Yaskawa INFORM job: DEMO_ROOF_SIDE_0625_3PAINT_2.JBI

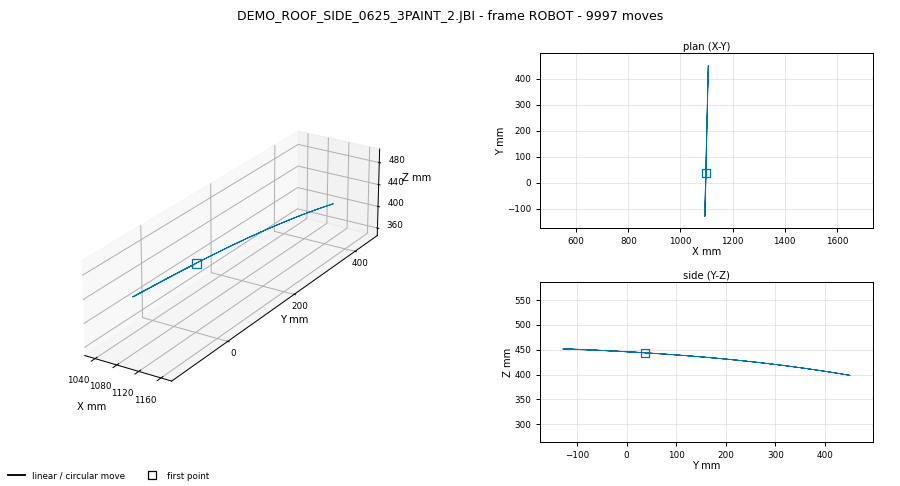
[picture p0: tool path of DEMO_ROOF_SIDE_0625_3PAINT_2.JBI in frame ROBOT, 9997 of 9997 moves have a stored position in this frame; points joined in program order, loops and branches not executed]
/JOB
//NAME DEMO_ROOF_SIDE_0625_3PAINT2
//POS
///NPOS 9997,0,0,0,0,0
///TOOL 0
///USER 0
///POSTYPE ROBOT
///RECTAN
///RCONF 1,0,0,0,0,0,0,0,0,0,0,0,0,0,0,0,0,0,0,0,0,0,0,0
C00000=1098.370,36.999,444.195,176.206,15.311,152.033
C00001=1098.365,36.749,444.210,176.204,15.310,152.034
C00002=1098.358,36.500,444.225,176.201,15.310,152.034
C00003=1098.353,36.250,444.240,176.199,15.308,152.034
C00004=1098.347,36.001,444.255,176.197,15.308,152.035
C00005=1098.341,35.751,444.271,176.195,15.307,152.035
C00006=1098.336,35.502,444.287,176.192,15.306,152.035
C00007=1098.329,35.252,444.302,176.190,15.306,152.036
C00008=1098.324,35.003,444.317,176.188,15.305,152.036
C00009=1098.318,34.753,444.332,176.185,15.304,152.036
C00010=1098.312,34.503,444.347,176.183,15.303,152.037
C00011=1098.307,34.255,444.362,176.181,15.303,152.037
C00012=1098.301,34.005,444.377,176.178,15.302,152.037
C00013=1098.296,33.755,444.393,176.176,15.301,152.038
C00014=1098.289,33.506,444.407,176.174,15.301,152.038
C00015=1098.284,33.256,444.423,176.172,15.300,152.038
C00016=1098.278,33.007,444.438,176.170,15.299,152.038
C00017=1098.273,32.758,444.453,176.167,15.298,152.039
C00018=1098.266,32.508,444.468,176.166,15.298,152.039
C00019=1098.261,32.258,444.484,176.163,15.296,152.039
C00020=1098.254,31.985,444.500,176.161,15.296,152.040
C00021=1098.248,31.711,444.517,176.158,15.295,152.040
C00022=1098.242,31.437,444.534,176.156,15.294,152.041
C00023=1098.236,31.164,444.550,176.153,15.293,152.041
C00024=1098.230,30.914,444.565,176.151,15.292,152.041
C00025=1098.224,30.665,444.580,176.149,15.292,152.041
C00026=1098.218,30.415,444.595,176.147,15.291,152.042
C00027=1098.213,30.166,444.610,176.145,15.290,152.042
C00028=1098.207,29.916,444.625,176.142,15.290,152.042
C00029=1098.202,29.667,444.639,176.140,15.288,152.043
C00030=1098.196,29.417,444.655,176.138,15.288,152.043
C00031=1098.190,29.168,444.669,176.136,15.287,152.043
C00032=1098.185,28.918,444.685,176.134,15.287,152.044
C00033=1098.179,28.669,444.699,176.131,15.285,152.044
C00034=1098.172,28.419,444.714,176.129,15.285,152.044
C00035=1098.167,28.170,444.730,176.127,15.284,152.045
C00036=1098.161,27.920,444.745,176.124,15.283,152.045
C00037=1098.156,27.671,444.760,176.123,15.282,152.045
C00038=1098.149,27.421,444.775,176.121,15.281,152.045
C00039=1098.144,27.172,444.789,176.118,15.281,152.046
C00040=1098.138,26.922,444.804,176.116,15.280,152.046
C00041=1098.133,26.673,444.819,176.114,15.279,152.046
C00042=1098.126,26.423,444.834,176.112,15.278,152.047
C00043=1098.121,26.174,444.849,176.110,15.278,152.047
C00044=1098.115,25.925,444.863,176.107,15.277,152.047
C00045=1098.109,25.675,444.878,176.105,15.276,152.048
C00046=1098.104,25.425,444.893,176.103,15.275,152.048
C00047=1098.098,25.176,444.908,176.100,15.274,152.048
C00048=1098.092,24.927,444.922,176.099,15.274,152.049
C00049=1098.086,24.677,444.938,176.097,15.273,152.049
C00050=1098.081,24.427,444.952,176.095,15.272,152.049
C00051=1098.075,24.178,444.967,176.092,15.271,152.049
C00052=1098.069,23.929,444.981,176.090,15.271,152.050
C00053=1098.063,23.679,444.997,176.088,15.270,152.050
C00054=1098.058,23.429,445.011,176.086,15.269,152.050
C00055=1098.052,23.180,445.025,176.084,15.268,152.051
C00056=1098.046,22.930,445.041,176.081,15.268,152.051
C00057=1098.040,22.681,445.055,176.080,15.267,152.051
C00058=1098.034,22.431,445.070,176.077,15.265,152.051
C00059=1098.029,22.182,445.084,176.075,15.265,152.052
C00060=1098.024,21.933,445.099,176.073,15.264,152.052
C00061=1098.017,21.682,445.114,176.071,15.264,152.052
C00062=1098.012,21.434,445.128,176.068,15.262,152.053
C00063=1098.005,21.184,445.143,176.066,15.262,152.053
C00064=1098.001,20.934,445.158,176.064,15.261,152.053
C00065=1097.995,20.685,445.172,176.063,15.260,152.053
C00066=1097.988,20.435,445.187,176.060,15.259,152.054
C00067=1097.983,20.186,445.201,176.058,15.258,152.054
C00068=1097.978,19.937,445.216,176.056,15.258,152.054
C00069=1097.972,19.687,445.231,176.054,15.257,152.055
C00070=1097.966,19.437,445.245,176.051,15.256,152.055
C00071=1097.960,19.188,445.260,176.049,15.255,152.055
C00072=1097.954,18.938,445.274,176.048,15.254,152.055
C00073=1097.948,18.689,445.288,176.046,15.254,152.056
C00074=1097.942,18.439,445.303,176.043,15.253,152.056
C00075=1097.937,18.190,445.318,176.041,15.252,152.056
C00076=1097.932,17.941,445.332,176.039,15.251,152.057
C00077=1097.925,17.690,445.347,176.037,15.251,152.057
C00078=1097.920,17.441,445.361,176.034,15.249,152.057
C00079=1097.914,17.192,445.375,176.033,15.248,152.057
C00080=1097.908,16.942,445.390,176.031,15.248,152.058
C00081=1097.902,16.693,445.404,176.028,15.247,152.058
C00082=1097.897,16.444,445.418,176.026,15.246,152.058
C00083=1097.891,16.193,445.433,176.024,15.245,152.059
C00084=1097.884,15.922,445.449,176.022,15.245,152.059
C00085=1097.878,15.649,445.465,176.019,15.243,152.059
C00086=1097.872,15.376,445.480,176.017,15.243,152.059
C00087=1097.866,15.104,445.495,176.015,15.241,152.060
C00088=1097.859,14.854,445.510,176.013,15.241,152.060
C00089=1097.855,14.605,445.525,176.011,15.240,152.060
C00090=1097.849,14.356,445.539,176.009,15.240,152.061
C00091=1097.843,14.106,445.553,176.006,15.238,152.061
C00092=1097.837,13.856,445.568,176.004,15.237,152.061
C00093=1097.831,13.607,445.581,176.002,15.237,152.061
C00094=1097.825,13.358,445.596,176.001,15.236,152.062
C00095=1097.819,13.108,445.610,175.999,15.235,152.062
C00096=1097.814,12.858,445.624,175.996,15.234,152.062
C00097=1097.808,12.609,445.639,175.994,15.234,152.063
C00098=1097.802,12.359,445.653,175.992,15.233,152.063
C00099=1097.796,12.110,445.667,175.990,15.232,152.063
C00100=1097.790,11.861,445.681,175.987,15.231,152.064
C00101=1097.784,11.610,445.696,175.986,15.230,152.064
C00102=1097.779,11.361,445.710,175.984,15.229,152.064
C00103=1097.773,11.112,445.724,175.982,15.229,152.064
C00104=1097.767,10.862,445.739,175.980,15.228,152.065
C00105=1097.761,10.613,445.753,175.977,15.227,152.065
C00106=1097.755,10.363,445.766,175.975,15.226,152.065
C00107=1097.749,10.114,445.781,175.973,15.225,152.065
C00108=1097.743,9.864,445.795,175.971,15.225,152.066
C00109=1097.738,9.614,445.809,175.969,15.224,152.066
C00110=1097.732,9.365,445.823,175.967,15.223,152.066
C00111=1097.726,9.115,445.838,175.965,15.222,152.067
C00112=1097.720,8.866,445.851,175.963,15.221,152.067
C00113=1097.715,8.616,445.865,175.961,15.221,152.067
C00114=1097.708,8.367,445.879,175.958,15.219,152.067
C00115=1097.702,8.117,445.893,175.957,15.219,152.068
C00116=1097.697,7.868,445.907,175.955,15.218,152.068
C00117=1097.691,7.618,445.921,175.953,15.217,152.068
C00118=1097.685,7.369,445.936,175.951,15.216,152.068
C00119=1097.679,7.119,445.950,175.948,15.215,152.069
C00120=1097.674,6.869,445.964,175.946,15.214,152.069
C00121=1097.668,6.620,445.977,175.944,15.214,152.069
C00122=1097.662,6.370,445.991,175.943,15.213,152.069
C00123=1097.656,6.121,446.006,175.941,15.212,152.070
C00124=1097.650,5.871,446.020,175.938,15.211,152.070
C00125=1097.645,5.622,446.034,175.936,15.210,152.070
C00126=1097.639,5.372,446.048,175.934,15.209,152.070
C00127=1097.633,5.123,446.061,175.932,15.209,152.071
C00128=1097.627,4.874,446.075,175.931,15.208,152.071
C00129=1097.621,4.623,446.090,175.928,15.207,152.071
C00130=1097.616,4.374,446.104,175.926,15.206,152.072
C00131=1097.610,4.124,446.117,175.924,15.205,152.072
C00132=1097.604,3.875,446.131,175.922,15.204,152.072
C00133=1097.599,3.625,446.145,175.920,15.204,152.072
C00134=1097.593,3.376,446.158,175.918,15.202,152.073
C00135=1097.588,3.126,446.172,175.916,15.202,152.073
C00136=1097.581,2.877,446.187,175.914,15.201,152.073
C00137=1097.575,2.627,446.200,175.912,15.200,152.073
C00138=1097.570,2.378,446.214,175.910,15.199,152.073
C00139=1097.564,2.128,446.228,175.908,15.198,152.074
C00140=1097.559,1.879,446.242,175.906,15.197,152.074
C00141=1097.553,1.629,446.255,175.904,15.196,152.074
C00142=1097.547,1.380,446.269,175.902,15.195,152.075
C00143=1097.541,1.130,446.283,175.900,15.195,152.075
C00144=1097.536,0.880,446.297,175.898,15.194,152.075
C00145=1097.529,0.631,446.311,175.896,15.193,152.075
C00146=1097.524,0.381,446.324,175.894,15.192,152.076
C00147=1097.518,0.132,446.338,175.892,15.191,152.076
C00148=1097.512,-0.139,446.354,175.890,15.190,152.076
C00149=1097.506,-0.409,446.368,175.887,15.189,152.076
C00150=1097.500,-0.679,446.383,175.886,15.188,152.077
C00151=1097.493,-0.949,446.398,175.884,15.188,152.077
C00152=1097.488,-1.199,446.411,175.881,15.186,152.077
C00153=1097.482,-1.448,446.425,175.879,15.185,152.077
C00154=1097.476,-1.699,446.440,175.878,15.184,152.078
C00155=1097.470,-1.948,446.453,175.876,15.184,152.078
C00156=1097.465,-2.198,446.466,175.874,15.183,152.078
C00157=1097.459,-2.448,446.480,175.871,15.182,152.078
C00158=1097.454,-2.697,446.494,175.869,15.181,152.079
C00159=1097.448,-2.946,446.507,175.867,15.180,152.079
C00160=1097.442,-3.196,446.521,175.866,15.179,152.079
C00161=1097.437,-3.446,446.535,175.864,15.178,152.079
C00162=1097.431,-3.695,446.548,175.862,15.177,152.079
C00163=1097.425,-3.944,446.562,175.859,15.176,152.080
C00164=1097.419,-4.194,446.575,175.858,15.175,152.080
C00165=1097.413,-4.443,446.589,175.856,15.175,152.080
C00166=1097.407,-4.693,446.602,175.854,15.174,152.081
C00167=1097.401,-4.943,446.616,175.852,15.173,152.081
C00168=1097.395,-5.193,446.629,175.850,15.172,152.081
C00169=1097.390,-5.442,446.643,175.847,15.171,152.081
C00170=1097.383,-5.692,446.656,175.845,15.170,152.082
C00171=1097.378,-5.941,446.670,175.844,15.170,152.082
C00172=1097.372,-6.190,446.683,175.842,15.169,152.082
C00173=1097.367,-6.441,446.696,175.840,15.168,152.082
C00174=1097.360,-6.690,446.710,175.838,15.167,152.082
C00175=1097.355,-6.939,446.724,175.836,15.166,152.083
C00176=1097.349,-7.189,446.737,175.834,15.165,152.083
C00177=1097.343,-7.438,446.751,175.832,15.164,152.083
C00178=1097.337,-7.688,446.763,175.830,15.163,152.084
C00179=1097.331,-7.937,446.777,175.828,15.163,152.084
C00180=1097.326,-8.187,446.790,175.826,15.162,152.084
C00181=1097.319,-8.436,446.804,175.824,15.161,152.084
C00182=1097.314,-8.686,446.817,175.822,15.161,152.085
C00183=1097.308,-8.936,446.830,175.820,15.159,152.085
C00184=1097.303,-9.185,446.844,175.818,15.158,152.085
C00185=1097.296,-9.435,446.857,175.816,15.157,152.085
C00186=1097.291,-9.685,446.870,175.814,15.157,152.085
C00187=1097.284,-9.935,446.884,175.813,15.156,152.086
C00188=1097.278,-10.184,446.897,175.811,15.155,152.086
C00189=1097.273,-10.434,446.911,175.809,15.154,152.086
C00190=1097.267,-10.683,446.923,175.806,15.153,152.087
C00191=1097.262,-10.932,446.937,175.805,15.152,152.087
C00192=1097.256,-11.182,446.950,175.803,15.151,152.087
C00193=1097.251,-11.432,446.964,175.801,15.150,152.087
C00194=1097.244,-11.681,446.977,175.799,15.150,152.087
C00195=1097.238,-11.930,446.990,175.797,15.149,152.088
C00196=1097.233,-12.180,447.003,175.795,15.148,152.088
C00197=1097.227,-12.430,447.017,175.794,15.147,152.088
C00198=1097.222,-12.680,447.030,175.791,15.146,152.088
C00199=1097.215,-12.929,447.043,175.789,15.145,152.089
C00200=1097.209,-13.178,447.056,175.787,15.144,152.089
C00201=1097.204,-13.429,447.069,175.785,15.143,152.089
C00202=1097.198,-13.678,447.083,175.783,15.143,152.089
C00203=1097.193,-13.928,447.096,175.782,15.142,152.089
C00204=1097.186,-14.177,447.109,175.780,15.141,152.090
C00205=1097.180,-14.427,447.122,175.778,15.140,152.090
C00206=1097.175,-14.677,447.135,175.775,15.139,152.090
C00207=1097.169,-14.926,447.149,175.773,15.138,152.091
C00208=1097.163,-15.176,447.161,175.772,15.137,152.091
C00209=1097.157,-15.426,447.175,175.770,15.136,152.091
C00210=1097.151,-15.675,447.188,175.768,15.135,152.091
C00211=1097.145,-15.925,447.201,175.766,15.135,152.091
C00212=1097.139,-16.194,447.215,175.764,15.134,152.092
C00213=1097.133,-16.462,447.229,175.762,15.133,152.092
C00214=1097.127,-16.731,447.243,175.760,15.132,152.092
C00215=1097.120,-16.999,447.257,175.758,15.131,152.092
C00216=1097.114,-17.249,447.270,175.756,15.130,152.093
C00217=1097.109,-17.498,447.284,175.754,15.129,152.093
C00218=1097.103,-17.748,447.296,175.752,15.128,152.093
C00219=1097.097,-17.997,447.309,175.750,15.127,152.093
C00220=1097.091,-18.247,447.322,175.748,15.126,152.094
C00221=1097.085,-18.497,447.335,175.746,15.126,152.094
C00222=1097.079,-18.747,447.348,175.744,15.125,152.094
C00223=1097.073,-18.997,447.361,175.743,15.124,152.094
C00224=1097.067,-19.246,447.374,175.741,15.123,152.094
C00225=1097.061,-19.496,447.387,175.739,15.122,152.095
C00226=1097.056,-19.744,447.400,175.737,15.122,152.095
C00227=1097.050,-19.994,447.412,175.735,15.121,152.095
C00228=1097.044,-20.244,447.426,175.733,15.120,152.096
C00229=1097.038,-20.494,447.439,175.731,15.118,152.096
C00230=1097.033,-20.743,447.451,175.729,15.118,152.096
C00231=1097.026,-20.993,447.464,175.727,15.117,152.096
C00232=1097.020,-21.243,447.477,175.725,15.116,152.096
C00233=1097.014,-21.492,447.490,175.723,15.115,152.097
C00234=1097.010,-21.741,447.503,175.722,15.114,152.097
C00235=1097.004,-21.991,447.516,175.720,15.114,152.097
C00236=1096.998,-22.241,447.529,175.718,15.113,152.097
C00237=1096.992,-22.490,447.541,175.716,15.112,152.098
C00238=1096.986,-22.740,447.554,175.714,15.111,152.098
C00239=1096.979,-22.990,447.567,175.713,15.110,152.098
C00240=1096.974,-23.239,447.580,175.710,15.109,152.098
C00241=1096.969,-23.489,447.593,175.708,15.108,152.098
C00242=1096.963,-23.738,447.606,175.706,15.107,152.099
C00243=1096.957,-23.988,447.618,175.704,15.107,152.099
C00244=1096.951,-24.238,447.631,175.703,15.105,152.099
C00245=1096.945,-24.488,447.644,175.701,15.105,152.099
C00246=1096.939,-24.736,447.656,175.699,15.104,152.100
C00247=1096.934,-24.986,447.669,175.697,15.103,152.100
C00248=1096.928,-25.236,447.682,175.696,15.102,152.100
C00249=1096.921,-25.485,447.695,175.694,15.101,152.100
C00250=1096.916,-25.735,447.707,175.692,15.101,152.100
C00251=1096.911,-25.985,447.720,175.690,15.100,152.101
C00252=1096.905,-26.235,447.733,175.688,15.099,152.101
C00253=1096.899,-26.484,447.746,175.686,15.097,152.101
C00254=1096.893,-26.734,447.759,175.684,15.097,152.101
C00255=1096.887,-26.984,447.771,175.682,15.096,152.102
C00256=1096.882,-27.233,447.783,175.680,15.095,152.102
C00257=1096.876,-27.483,447.796,175.679,15.094,152.102
C00258=1096.870,-27.732,447.809,175.677,15.093,152.102
C00259=1096.864,-27.982,447.822,175.675,15.093,152.103
C00260=1096.858,-28.232,447.834,175.673,15.092,152.103
C00261=1096.851,-28.481,447.846,175.671,15.091,152.103
C00262=1096.846,-28.731,447.858,175.669,15.090,152.103
C00263=1096.840,-28.980,447.872,175.668,15.089,152.103
C00264=1096.834,-29.230,447.884,175.666,15.088,152.104
C00265=1096.828,-29.480,447.897,175.664,15.088,152.104
C00266=1096.822,-29.729,447.909,175.662,15.087,152.104
C00267=1096.817,-29.979,447.921,175.660,15.086,152.104
C00268=1096.811,-30.229,447.934,175.658,15.085,152.105
C00269=1096.805,-30.478,447.947,175.657,15.084,152.105
C00270=1096.799,-30.728,447.960,175.655,15.084,152.105
C00271=1096.793,-30.977,447.972,175.653,15.083,152.105
C00272=1096.787,-31.226,447.984,175.650,15.082,152.106
C00273=1096.781,-31.476,447.997,175.649,15.080,152.106
C00274=1096.775,-31.726,448.009,175.647,15.080,152.106
C00275=1096.769,-31.976,448.022,175.645,15.079,152.106
C00276=1096.763,-32.244,448.035,175.643,15.078,152.106
C00277=1096.757,-32.511,448.048,175.641,15.078,152.107
C00278=1096.750,-32.780,448.062,175.639,15.077,152.107
C00279=1096.744,-33.047,448.076,175.638,15.076,152.107
C00280=1096.737,-33.297,448.088,175.636,15.075,152.107
C00281=1096.732,-33.546,448.100,175.634,15.074,152.108
C00282=1096.726,-33.796,448.112,175.632,15.073,152.108
C00283=1096.720,-34.046,448.125,175.629,15.072,152.108
C00284=1096.714,-34.296,448.137,175.628,15.071,152.108
C00285=1096.709,-34.545,448.150,175.626,15.070,152.109
C00286=1096.702,-34.794,448.162,175.624,15.069,152.109
C00287=1096.697,-35.044,448.174,175.622,15.069,152.109
C00288=1096.691,-35.294,448.186,175.620,15.068,152.109
C00289=1096.685,-35.543,448.199,175.619,15.067,152.109
C00290=1096.679,-35.793,448.211,175.617,15.066,152.110
C00291=1096.674,-36.042,448.224,175.615,15.065,152.110
C00292=1096.668,-36.292,448.236,175.613,15.064,152.110
C00293=1096.662,-36.542,448.248,175.611,15.063,152.110
C00294=1096.657,-36.792,448.260,175.609,15.063,152.111
C00295=1096.651,-37.042,448.272,175.608,15.062,152.111
C00296=1096.645,-37.292,448.285,175.606,15.061,152.111
C00297=1096.639,-37.541,448.297,175.604,15.060,152.111
C00298=1096.633,-37.790,448.309,175.602,15.059,152.111
C00299=1096.627,-38.040,448.321,175.600,15.059,152.112
C00300=1096.622,-38.289,448.334,175.599,15.058,152.112
C00301=1096.616,-38.539,448.346,175.597,15.057,152.112
C00302=1096.609,-38.789,448.358,175.595,15.056,152.112
C00303=1096.604,-39.038,448.370,175.593,15.055,152.113
C00304=1096.598,-39.288,448.383,175.591,15.055,152.113
C00305=1096.592,-39.538,448.394,175.590,15.053,152.113
C00306=1096.586,-39.787,448.406,175.588,15.053,152.113
C00307=1096.580,-40.037,448.419,175.586,15.052,152.113
C00308=1096.574,-40.287,448.431,175.584,15.051,152.114
C00309=1096.568,-40.537,448.443,175.582,15.050,152.114
C00310=1096.562,-40.786,448.455,175.580,15.050,152.114
C00311=1096.556,-41.035,448.467,175.579,15.049,152.114
C00312=1096.550,-41.286,448.479,175.577,15.048,152.115
C00313=1096.545,-41.535,448.491,175.575,15.047,152.115
C00314=1096.538,-41.785,448.503,175.573,15.046,152.115
C00315=1096.533,-42.034,448.516,175.571,15.046,152.115
C00316=1096.526,-42.283,448.528,175.570,15.044,152.116
C00317=1096.521,-42.534,448.539,175.568,15.044,152.116
C00318=1096.515,-42.783,448.552,175.566,15.043,152.116
C00319=1096.509,-43.033,448.564,175.564,15.042,152.116
C00320=1096.503,-43.282,448.576,175.562,15.042,152.117
C00321=1096.497,-43.531,448.588,175.561,15.040,152.117
C00322=1096.491,-43.782,448.600,175.559,15.040,152.117
C00323=1096.485,-44.032,448.612,175.557,15.039,152.117
C00324=1096.479,-44.281,448.624,175.555,15.038,152.117
C00325=1096.473,-44.530,448.636,175.553,15.037,152.118
C00326=1096.468,-44.780,448.647,175.551,15.036,152.118
C00327=1096.462,-45.030,448.660,175.550,15.036,152.118
C00328=1096.456,-45.280,448.672,175.548,15.035,152.118
C00329=1096.450,-45.529,448.683,175.546,15.034,152.119
C00330=1096.444,-45.779,448.696,175.545,15.034,152.119
C00331=1096.438,-46.028,448.707,175.543,15.033,152.119
C00332=1096.432,-46.278,448.720,175.541,15.032,152.119
C00333=1096.426,-46.528,448.731,175.539,15.031,152.119
C00334=1096.420,-46.777,448.743,175.537,15.031,152.120
C00335=1096.414,-47.027,448.755,175.536,15.029,152.120
C00336=1096.409,-47.277,448.767,175.534,15.029,152.120
C00337=1096.403,-47.526,448.779,175.532,15.028,152.120
C00338=1096.397,-47.775,448.791,175.530,15.027,152.121
C00339=1096.391,-48.026,448.803,175.529,15.026,152.121
C00340=1096.385,-48.293,448.815,175.527,15.025,152.121
C00341=1096.378,-48.562,448.828,175.525,15.025,152.121
C00342=1096.372,-48.830,448.840,175.523,15.024,152.121
C00343=1096.366,-49.098,448.853,175.520,15.023,152.122
C00344=1096.360,-49.348,448.866,175.518,15.022,152.122
C00345=1096.354,-49.598,448.877,175.518,15.021,152.122
C00346=1096.348,-49.848,448.889,175.516,15.021,152.122
C00347=1096.343,-50.097,448.900,175.514,15.020,152.123
C00348=1096.337,-50.347,448.913,175.512,15.019,152.123
C00349=1096.331,-50.596,448.924,175.510,15.018,152.123
C00350=1096.324,-50.846,448.935,175.509,15.017,152.123
C00351=1096.319,-51.096,448.948,175.507,15.017,152.123
C00352=1096.313,-51.345,448.959,175.505,15.016,152.124
C00353=1096.306,-51.595,448.971,175.503,15.015,152.124
C00354=1096.301,-51.845,448.982,175.501,15.014,152.124
C00355=1096.294,-52.094,448.994,175.499,15.014,152.125
C00356=1096.288,-52.344,449.006,175.498,15.012,152.125
C00357=1096.283,-52.594,449.018,175.496,15.012,152.125
C00358=1096.276,-52.843,449.030,175.494,15.011,152.125
C00359=1096.270,-53.093,449.041,175.492,15.010,152.125
C00360=1096.264,-53.342,449.052,175.490,15.010,152.126
C00361=1096.259,-53.592,449.064,175.489,15.009,152.126
C00362=1096.252,-53.842,449.076,175.487,15.009,152.126
C00363=1096.246,-54.092,449.087,175.485,15.008,152.126
C00364=1096.240,-54.341,449.099,175.484,15.007,152.127
C00365=1096.234,-54.591,449.111,175.482,15.006,152.127
C00366=1096.228,-54.840,449.122,175.480,15.005,152.127
C00367=1096.222,-55.090,449.133,175.478,15.005,152.127
C00368=1096.216,-55.340,449.146,175.476,15.004,152.128
C00369=1096.210,-55.590,449.157,175.474,15.003,152.128
C00370=1096.204,-55.839,449.168,175.472,15.003,152.128
C00371=1096.198,-56.089,449.180,175.471,15.001,152.128
C00372=1096.193,-56.339,449.191,175.469,15.001,152.128
C00373=1096.186,-56.588,449.203,175.468,15.001,152.129
C00374=1096.180,-56.838,449.214,175.466,15.000,152.129
C00375=1096.174,-57.087,449.226,175.464,14.999,152.129
C00376=1096.168,-57.337,449.237,175.462,14.998,152.129
C00377=1096.162,-57.587,449.249,175.460,14.998,152.130
C00378=1096.156,-57.836,449.260,175.459,14.996,152.130
C00379=1096.150,-58.086,449.272,175.457,14.996,152.130
C00380=1096.144,-58.336,449.282,175.455,14.995,152.130
C00381=1096.138,-58.586,449.295,175.453,14.994,152.131
C00382=1096.133,-58.835,449.306,175.451,14.994,152.131
C00383=1096.126,-59.085,449.318,175.450,14.993,152.131
C00384=1096.120,-59.334,449.329,175.448,14.993,152.131
C00385=1096.114,-59.584,449.340,175.446,14.992,152.131
C00386=1096.109,-59.834,449.352,175.445,14.991,152.132
C00387=1096.102,-60.084,449.363,175.443,14.990,152.132
C00388=1096.096,-60.333,449.374,175.441,14.989,152.132
C00389=1096.090,-60.583,449.386,175.439,14.989,152.133
C00390=1096.084,-60.832,449.397,175.437,14.988,152.133
C00391=1096.079,-61.082,449.409,175.435,14.987,152.133
C00392=1096.072,-61.332,449.420,175.434,14.987,152.133
C00393=1096.067,-61.581,449.431,175.432,14.986,152.133
C00394=1096.060,-61.831,449.443,175.431,14.985,152.134
C00395=1096.055,-62.081,449.453,175.429,14.985,152.134
C00396=1096.048,-62.330,449.465,175.427,14.984,152.134
C00397=1096.043,-62.580,449.477,175.425,14.983,152.134
C00398=1096.037,-62.830,449.488,175.423,14.982,152.135
C00399=1096.031,-63.080,449.499,175.421,14.981,152.135
C00400=1096.025,-63.329,449.511,175.420,14.981,152.135
C00401=1096.019,-63.579,449.522,175.418,14.980,152.135
C00402=1096.013,-63.828,449.533,175.417,14.980,152.136
C00403=1096.007,-64.078,449.544,175.415,14.979,152.136
C00404=1096.000,-64.348,449.557,175.413,14.978,152.136
C00405=1095.994,-64.618,449.569,175.411,14.977,152.136
C00406=1095.988,-64.887,449.581,175.409,14.976,152.136
C00407=1095.982,-65.157,449.593,175.407,14.976,152.137
C00408=1095.976,-65.406,449.604,175.406,14.975,152.137
C00409=1095.969,-65.656,449.616,175.404,14.974,152.137
C00410=1095.964,-65.905,449.626,175.402,14.973,152.138
C00411=1095.957,-66.155,449.638,175.400,14.973,152.138
C00412=1095.951,-66.405,449.649,175.399,14.973,152.138
C00413=1095.946,-66.655,449.660,175.397,14.971,152.138
C00414=1095.940,-66.904,449.672,175.395,14.971,152.138
C00415=1095.934,-67.154,449.683,175.394,14.970,152.139
C00416=1095.928,-67.403,449.694,175.392,14.969,152.139
C00417=1095.922,-67.653,449.705,175.390,14.969,152.139
C00418=1095.916,-67.903,449.716,175.388,14.968,152.139
C00419=1095.910,-68.152,449.727,175.387,14.967,152.139
C00420=1095.904,-68.403,449.738,175.385,14.967,152.140
C00421=1095.898,-68.652,449.749,175.383,14.966,152.140
C00422=1095.893,-68.902,449.760,175.381,14.965,152.140
C00423=1095.886,-69.151,449.772,175.380,14.964,152.141
C00424=1095.881,-69.401,449.783,175.378,14.964,152.141
C00425=1095.875,-69.650,449.794,175.377,14.964,152.141
C00426=1095.870,-69.900,449.805,175.375,14.962,152.141
C00427=1095.863,-70.150,449.816,175.373,14.962,152.141
C00428=1095.857,-70.400,449.827,175.371,14.961,152.142
C00429=1095.852,-70.649,449.838,175.369,14.960,152.142
C00430=1095.845,-70.899,449.849,175.367,14.960,152.142
C00431=1095.840,-71.149,449.860,175.366,14.959,152.142
C00432=1095.834,-71.398,449.871,175.364,14.959,152.143
C00433=1095.828,-71.648,449.882,175.363,14.958,152.143
C00434=1095.822,-71.898,449.893,175.361,14.957,152.143
C00435=1095.816,-72.147,449.904,175.359,14.956,152.143
C00436=1095.810,-72.397,449.915,175.357,14.955,152.144
C00437=1095.805,-72.646,449.926,175.355,14.955,152.144
C00438=1095.798,-72.897,449.937,175.354,14.955,152.144
C00439=1095.793,-73.146,449.948,175.353,14.953,152.144
C00440=1095.787,-73.396,449.959,175.351,14.953,152.144
C00441=1095.781,-73.645,449.969,175.349,14.952,152.145
C00442=1095.775,-73.895,449.981,175.347,14.951,152.145
C00443=1095.769,-74.145,449.992,175.346,14.951,152.145
C00444=1095.763,-74.394,450.002,175.344,14.950,152.145
C00445=1095.757,-74.644,450.014,175.342,14.950,152.146
C00446=1095.751,-74.894,450.025,175.340,14.949,152.146
C00447=1095.745,-75.143,450.035,175.338,14.948,152.146
C00448=1095.740,-75.393,450.046,175.337,14.948,152.146
C00449=1095.733,-75.643,450.058,175.336,14.947,152.147
C00450=1095.728,-75.893,450.068,175.334,14.946,152.147
C00451=1095.721,-76.142,450.078,175.332,14.946,152.147
C00452=1095.715,-76.393,450.089,175.330,14.945,152.147
C00453=1095.709,-76.642,450.100,175.329,14.945,152.148
C00454=1095.704,-76.892,450.111,175.327,14.944,152.148
C00455=1095.698,-77.141,450.122,175.325,14.943,152.148
C00456=1095.692,-77.391,450.133,175.323,14.943,152.148
C00457=1095.685,-77.640,450.143,175.321,14.942,152.149
C00458=1095.679,-77.890,450.154,175.320,14.942,152.149
C00459=1095.674,-78.139,450.165,175.318,14.941,152.149
C00460=1095.668,-78.390,450.176,175.316,14.940,152.149
C00461=1095.662,-78.640,450.187,175.315,14.940,152.150
C00462=1095.656,-78.889,450.197,175.313,14.939,152.150
C00463=1095.650,-79.138,450.208,175.312,14.939,152.150
C00464=1095.643,-79.389,450.219,175.310,14.938,152.150
C00465=1095.637,-79.638,450.230,175.308,14.937,152.151
C00466=1095.632,-79.888,450.241,175.306,14.936,152.151
C00467=1095.626,-80.138,450.251,175.305,14.936,152.151
C00468=1095.619,-80.409,450.262,175.303,14.936,152.151
C00469=1095.612,-80.681,450.274,175.301,14.935,152.152
C00470=1095.606,-80.953,450.286,175.299,14.934,152.152
C00471=1095.599,-81.224,450.298,175.297,14.934,152.152
C00472=1095.593,-81.474,450.307,175.295,14.933,152.153
C00473=1095.587,-81.724,450.318,175.293,14.932,152.153
C00474=1095.581,-81.974,450.330,175.292,14.932,152.153
C00475=1095.574,-82.223,450.340,175.290,14.932,152.153
C00476=1095.569,-82.473,450.351,175.289,14.931,152.154
C00477=1095.563,-82.723,450.361,175.287,14.930,152.154
C00478=1095.556,-82.973,450.372,175.286,14.930,152.154
C00479=1095.550,-83.222,450.382,175.284,14.929,152.154
C00480=1095.544,-83.471,450.393,175.282,14.929,152.155
C00481=1095.539,-83.721,450.403,175.280,14.928,152.155
C00482=1095.532,-83.972,450.414,175.279,14.928,152.155
C00483=1095.526,-84.221,450.424,175.277,14.927,152.155
C00484=1095.520,-84.470,450.435,175.275,14.926,152.156
C00485=1095.515,-84.720,450.445,175.273,14.926,152.156
C00486=1095.508,-84.970,450.456,175.272,14.926,152.156
C00487=1095.502,-85.220,450.467,175.270,14.925,152.156
C00488=1095.496,-85.470,450.477,175.268,14.924,152.157
C00489=1095.490,-85.719,450.487,175.266,14.923,152.157
C00490=1095.484,-85.968,450.498,175.265,14.923,152.157
C00491=1095.477,-86.219,450.508,175.263,14.923,152.157
C00492=1095.472,-86.468,450.519,175.262,14.922,152.158
C00493=1095.465,-86.718,450.529,175.260,14.921,152.158
C00494=1095.460,-86.968,450.540,175.259,14.921,152.158
C00495=1095.454,-87.217,450.550,175.256,14.921,152.159
C00496=1095.447,-87.466,450.561,175.254,14.920,152.159
C00497=1095.441,-87.717,450.571,175.253,14.919,152.159
C00498=1095.435,-87.966,450.582,175.251,14.919,152.159
C00499=1095.429,-88.216,450.592,175.250,14.919,152.160
C00500=1095.423,-88.466,450.602,175.248,14.918,152.160
C00501=1095.417,-88.715,450.613,175.247,14.918,152.160
C00502=1095.412,-88.965,450.623,175.245,14.917,152.160
C00503=1095.405,-89.215,450.634,175.243,14.916,152.161
C00504=1095.399,-89.465,450.645,175.241,14.916,152.161
C00505=1095.393,-89.714,450.654,175.240,14.916,152.161
C00506=1095.387,-89.964,450.665,175.238,14.915,152.161
C00507=1095.381,-90.214,450.675,175.236,14.914,152.162
C00508=1095.375,-90.463,450.685,175.235,14.914,152.162
C00509=1095.369,-90.712,450.696,175.233,14.913,152.162
C00510=1095.363,-90.963,450.706,175.231,14.913,152.162
C00511=1095.356,-91.212,450.716,175.229,14.912,152.163
C00512=1095.351,-91.463,450.727,175.228,14.912,152.163
C00513=1095.345,-91.712,450.738,175.226,14.911,152.163
C00514=1095.339,-91.962,450.747,175.224,14.910,152.163
C00515=1095.333,-92.211,450.758,175.223,14.910,152.164
C00516=1095.327,-92.461,450.768,175.221,14.910,152.164
C00517=1095.321,-92.711,450.778,175.219,14.909,152.164
C00518=1095.315,-92.960,450.788,175.217,14.909,152.165
C00519=1095.309,-93.211,450.799,175.216,14.909,152.165
C00520=1095.303,-93.460,450.809,175.214,14.908,152.165
C00521=1095.297,-93.710,450.820,175.212,14.907,152.165
C00522=1095.291,-93.960,450.829,175.211,14.907,152.166
C00523=1095.285,-94.209,450.840,175.209,14.906,152.166
C00524=1095.279,-94.459,450.850,175.208,14.906,152.166
C00525=1095.273,-94.708,450.861,175.206,14.906,152.166
C00526=1095.267,-94.958,450.870,175.205,14.905,152.167
C00527=1095.261,-95.208,450.881,175.203,14.904,152.167
C00528=1095.255,-95.458,450.891,175.202,14.904,152.167
C00529=1095.249,-95.708,450.901,175.200,14.903,152.167
C00530=1095.243,-95.957,450.911,175.198,14.903,152.168
C00531=1095.238,-96.207,450.921,175.196,14.902,152.168
C00532=1095.231,-96.481,450.932,175.194,14.902,152.168
C00533=1095.224,-96.755,450.943,175.193,14.902,152.169
C00534=1095.218,-97.028,450.955,175.191,14.901,152.169
C00535=1095.211,-97.302,450.966,175.189,14.900,152.169
C00536=1095.204,-97.553,450.976,175.187,14.899,152.169
C00537=1095.199,-97.803,450.986,175.186,14.899,152.170
C00538=1095.192,-98.052,450.997,175.184,14.899,152.170
C00539=1095.186,-98.302,451.006,175.182,14.898,152.170
C00540=1095.180,-98.551,451.017,175.181,14.898,152.170
C00541=1095.174,-98.801,451.027,175.179,14.898,152.171
C00542=1095.168,-99.051,451.036,175.177,14.897,152.171
C00543=1095.162,-99.300,451.047,175.176,14.897,152.171
C00544=1095.156,-99.550,451.057,175.173,14.897,152.172
C00545=1095.150,-99.800,451.066,175.172,14.896,152.172
C00546=1095.144,-100.050,451.077,175.170,14.896,152.172
C00547=1095.138,-100.299,451.087,175.169,14.895,152.172
C00548=1095.132,-100.549,451.096,175.167,14.894,152.173
C00549=1095.125,-100.798,451.106,175.166,14.894,152.173
C00550=1095.119,-101.049,451.117,175.163,14.894,152.173
C00551=1095.113,-101.299,451.126,175.162,14.894,152.174
C00552=1095.107,-101.548,451.137,175.160,14.893,152.174
C00553=1095.101,-101.798,451.147,175.159,14.893,152.174
C00554=1095.095,-102.048,451.157,175.157,14.892,152.174
C00555=1095.089,-102.297,451.167,175.156,14.892,152.175
C00556=1095.083,-102.547,451.176,175.153,14.892,152.175
C00557=1095.077,-102.797,451.187,175.152,14.891,152.175
C00558=1095.071,-103.047,451.196,175.150,14.891,152.176
C00559=1095.064,-103.296,451.206,175.148,14.890,152.176
C00560=1095.058,-103.546,451.216,175.147,14.890,152.176
C00561=1095.053,-103.796,451.226,175.145,14.890,152.176
C00562=1095.046,-104.045,451.236,175.144,14.890,152.177
C00563=1095.040,-104.295,451.246,175.142,14.889,152.177
C00564=1095.034,-104.545,451.256,175.140,14.888,152.177
C00565=1095.029,-104.795,451.266,175.139,14.888,152.177
C00566=1095.022,-105.045,451.275,175.137,14.888,152.178
C00567=1095.016,-105.294,451.286,175.135,14.887,152.178
C00568=1095.010,-105.544,451.295,175.134,14.887,152.178
C00569=1095.004,-105.794,451.305,175.132,14.886,152.179
C00570=1094.998,-106.044,451.315,175.131,14.886,152.179
C00571=1094.992,-106.293,451.325,175.129,14.886,152.179
C00572=1094.986,-106.543,451.335,175.127,14.885,152.180
C00573=1094.979,-106.792,451.344,175.126,14.885,152.180
C00574=1094.974,-107.042,451.354,175.124,14.885,152.180
C00575=1094.968,-107.292,451.364,175.122,14.884,152.180
C00576=1094.962,-107.542,451.374,175.121,14.884,152.181
C00577=1094.955,-107.791,451.384,175.119,14.884,152.181
C00578=1094.949,-108.041,451.393,175.118,14.884,152.181
C00579=1094.943,-108.291,451.403,175.116,14.883,152.181
C00580=1094.937,-108.541,451.413,175.113,14.883,152.182
C00581=1094.931,-108.791,451.423,175.112,14.882,152.182
C00582=1094.925,-109.041,451.432,175.110,14.882,152.182
C00583=1094.918,-109.290,451.443,175.109,14.882,152.183
C00584=1094.912,-109.540,451.452,175.107,14.881,152.183
C00585=1094.906,-109.789,451.462,175.105,14.881,152.183
C00586=1094.900,-110.039,451.471,175.104,14.881,152.184
C00587=1094.894,-110.289,451.481,175.102,14.880,152.184
C00588=1094.888,-110.539,451.490,175.101,14.880,152.184
C00589=1094.881,-110.788,451.500,175.099,14.880,152.184
C00590=1094.876,-111.038,451.509,175.097,14.879,152.185
C00591=1094.870,-111.287,451.519,175.096,14.879,152.185
C00592=1094.864,-111.537,451.530,175.094,14.879,152.185
C00593=1094.858,-111.787,451.539,175.093,14.879,152.186
C00594=1094.852,-112.036,451.549,175.090,14.878,152.186
C00595=1094.845,-112.286,451.558,175.089,14.878,152.186
C00596=1094.839,-112.551,451.568,175.087,14.878,152.187
C00597=1094.833,-112.816,451.579,175.085,14.877,152.187
C00598=1094.826,-113.081,451.588,175.084,14.877,152.187
C00599=1094.820,-113.345,451.598,175.082,14.877,152.187
C00600=1094.813,-113.595,451.608,175.080,14.876,152.188
C00601=1094.807,-113.844,451.618,175.079,14.876,152.188
C00602=1094.801,-114.094,451.628,175.077,14.876,152.188
C00603=1094.795,-114.344,451.637,175.076,14.876,152.189
C00604=1094.788,-114.594,451.647,175.074,14.875,152.189
C00605=1094.782,-114.844,451.656,175.072,14.875,152.189
C00606=1094.776,-115.093,451.666,175.070,14.875,152.190
C00607=1094.770,-115.343,451.675,175.068,14.874,152.190
C00608=1094.764,-115.593,451.685,175.067,14.874,152.190
C00609=1094.758,-115.843,451.695,175.065,14.874,152.191
C00610=1094.751,-116.093,451.704,175.064,14.874,152.191
C00611=1094.746,-116.342,451.713,175.062,14.873,152.191
C00612=1094.740,-116.591,451.723,175.061,14.874,152.192
C00613=1094.733,-116.841,451.733,175.059,14.873,152.192
C00614=1094.728,-117.092,451.741,175.057,14.872,152.192
C00615=1094.721,-117.341,451.751,175.055,14.873,152.192
C00616=1094.715,-117.591,451.761,175.054,14.872,152.193
C00617=1094.709,-117.841,451.770,175.052,14.872,152.193
C00618=1094.703,-118.091,451.780,175.050,14.872,152.193
C00619=1094.697,-118.341,451.789,175.049,14.871,152.194
C00620=1094.691,-118.590,451.799,175.047,14.871,152.194
C00621=1094.684,-118.840,451.808,175.046,14.871,152.194
C00622=1094.679,-119.089,451.818,175.044,14.870,152.195
C00623=1094.672,-119.339,451.827,175.043,14.871,152.195
C00624=1094.666,-119.589,451.836,175.041,14.870,152.195
C00625=1094.660,-119.838,451.846,175.038,14.870,152.196
C00626=1094.653,-120.088,451.855,175.037,14.870,152.196
C00627=1094.647,-120.339,451.864,175.035,14.869,152.196
C00628=1094.641,-120.588,451.874,175.034,14.870,152.197
C00629=1094.635,-120.838,451.883,175.032,14.869,152.197
C00630=1094.630,-121.087,451.892,175.031,14.869,152.197
C00631=1094.623,-121.337,451.902,175.029,14.869,152.197
C00632=1094.616,-121.587,451.911,175.028,14.868,152.198
C00633=1094.610,-121.836,451.921,175.025,14.868,152.198
C00634=1094.604,-122.086,451.930,175.024,14.868,152.198
C00635=1094.598,-122.337,451.939,175.022,14.868,152.199
C00636=1094.592,-122.586,451.948,175.021,14.868,152.199
C00637=1094.587,-122.835,451.958,175.019,14.867,152.199
C00638=1094.580,-123.085,451.967,175.018,14.868,152.200
C00639=1094.573,-123.335,451.976,175.016,14.867,152.200
C00640=1094.567,-123.585,451.986,175.014,14.867,152.200
C00641=1094.561,-123.835,451.995,175.013,14.867,152.201
C00642=1094.555,-124.085,452.004,175.011,14.867,152.201
C00643=1094.549,-124.335,452.014,175.009,14.866,152.201
C00644=1094.544,-124.584,452.023,175.008,14.866,152.201
C00645=1094.537,-124.833,452.032,175.006,14.866,152.202
C00646=1094.531,-125.084,452.041,175.005,14.866,152.202
C00647=1094.525,-125.333,452.050,175.003,14.866,152.203
C00648=1094.518,-125.583,452.060,175.001,14.866,152.203
C00649=1094.511,-125.833,452.069,174.999,14.865,152.203
C00650=1094.506,-126.082,452.077,174.998,14.865,152.203
C00651=1094.500,-126.332,452.087,174.996,14.865,152.204
C00652=1094.494,-126.582,452.097,174.995,14.865,152.204
C00653=1094.487,-126.831,452.106,174.993,14.865,152.205
C00654=1094.481,-127.082,452.114,174.992,14.865,152.205
C00655=1094.475,-127.332,452.124,174.989,14.864,152.205
C00656=1094.468,-127.593,452.133,174.987,14.864,152.205
C00657=1094.462,-127.852,452.143,174.986,14.864,152.206
C00658=1094.456,-128.114,452.153,174.984,14.863,152.206
C00659=1094.457,-128.373,452.165,174.983,14.861,152.206
C00660=1094.050,-128.393,452.052,174.938,14.970,152.237
C00661=1094.047,-128.135,452.039,174.939,14.972,152.237
C00662=1094.054,-127.874,452.030,174.941,14.973,152.237
C00663=1094.060,-127.614,452.021,174.942,14.973,152.236
C00664=1094.067,-127.354,452.011,174.944,14.973,152.236
C00665=1094.072,-127.103,452.002,174.947,14.974,152.235
C00666=1094.079,-126.854,451.993,174.948,14.974,152.235
C00667=1094.086,-126.604,451.984,174.950,14.974,152.235
C00668=1094.092,-126.354,451.974,174.951,14.974,152.235
C00669=1094.097,-126.105,451.966,174.953,14.975,152.234
C00670=1094.104,-125.855,451.957,174.954,14.974,152.234
C00671=1094.110,-125.605,451.947,174.956,14.975,152.234
C00672=1094.116,-125.356,451.938,174.958,14.975,152.233
C00673=1094.122,-125.106,451.928,174.959,14.975,152.233
C00674=1094.129,-124.856,451.920,174.961,14.975,152.233
C00675=1094.135,-124.607,451.910,174.963,14.975,152.232
C00676=1094.141,-124.357,451.901,174.964,14.976,152.232
C00677=1094.147,-124.107,451.891,174.966,14.976,152.232
C00678=1094.153,-123.856,451.882,174.967,14.976,152.231
C00679=1094.159,-123.607,451.873,174.969,14.976,152.231
C00680=1094.166,-123.357,451.864,174.971,14.976,152.231
C00681=1094.171,-123.108,451.855,174.972,14.977,152.231
C00682=1094.178,-122.858,451.845,174.974,14.976,152.230
C00683=1094.184,-122.609,451.836,174.976,14.977,152.230
C00684=1094.190,-122.358,451.827,174.977,14.977,152.230
C00685=1094.196,-122.108,451.817,174.979,14.977,152.229
C00686=1094.202,-121.859,451.808,174.980,14.978,152.229
C00687=1094.209,-121.609,451.799,174.982,14.978,152.229
C00688=1094.214,-121.360,451.789,174.983,14.978,152.228
C00689=1094.221,-121.110,451.780,174.985,14.978,152.228
C00690=1094.227,-120.860,451.770,174.988,14.979,152.228
C00691=1094.233,-120.610,451.761,174.989,14.979,152.227
C00692=1094.239,-120.360,451.752,174.991,14.979,152.227
C00693=1094.245,-120.110,451.742,174.992,14.979,152.227
C00694=1094.251,-119.861,451.733,174.994,14.980,152.226
C00695=1094.258,-119.611,451.724,174.995,14.980,152.226
C00696=1094.264,-119.362,451.715,174.997,14.980,152.226
C00697=1094.270,-119.112,451.705,174.998,14.980,152.226
C00698=1094.276,-118.862,451.695,175.001,14.980,152.225
C00699=1094.282,-118.613,451.686,175.002,14.980,152.225
C00700=1094.288,-118.363,451.676,175.004,14.981,152.225
C00701=1094.294,-118.112,451.667,175.006,14.981,152.224
C00702=1094.300,-117.863,451.658,175.007,14.981,152.224
C00703=1094.307,-117.613,451.648,175.009,14.982,152.224
C00704=1094.313,-117.363,451.639,175.010,14.982,152.224
C00705=1094.318,-117.114,451.630,175.012,14.982,152.223
C00706=1094.324,-116.864,451.620,175.013,14.983,152.223
C00707=1094.331,-116.614,451.610,175.015,14.983,152.223
C00708=1094.337,-116.364,451.601,175.016,14.983,152.222
C00709=1094.343,-116.115,451.591,175.018,14.983,152.222
C00710=1094.350,-115.865,451.582,175.020,14.984,152.222
C00711=1094.356,-115.615,451.573,175.022,14.984,152.221
C00712=1094.362,-115.366,451.563,175.024,14.984,152.221
C00713=1094.368,-115.116,451.554,175.025,14.985,152.221
C00714=1094.375,-114.866,451.544,175.027,14.985,152.220
C00715=1094.381,-114.616,451.535,175.028,14.985,152.220
C00716=1094.387,-114.366,451.525,175.030,14.986,152.220
C00717=1094.393,-114.117,451.515,175.032,14.986,152.220
C00718=1094.399,-113.867,451.506,175.033,14.986,152.219
C00719=1094.404,-113.617,451.496,175.035,14.987,152.219
C00720=1094.410,-113.368,451.486,175.036,14.987,152.219
C00721=1094.417,-113.102,451.476,175.038,14.987,152.218
C00722=1094.423,-112.837,451.466,175.040,14.988,152.218
C00723=1094.430,-112.572,451.456,175.041,14.988,152.218
C00724=1094.437,-112.307,451.445,175.043,14.988,152.218
C00725=1094.443,-112.057,451.436,175.046,14.989,152.217
C00726=1094.449,-111.807,451.426,175.047,14.989,152.217
C00727=1094.455,-111.557,451.416,175.049,14.989,152.217
C00728=1094.461,-111.308,451.407,175.050,14.989,152.216
C00729=1094.468,-111.058,451.397,175.052,14.990,152.216
C00730=1094.474,-110.808,451.388,175.054,14.990,152.216
C00731=1094.479,-110.559,451.379,175.055,14.990,152.215
C00732=1094.485,-110.309,451.369,175.057,14.991,152.215
C00733=1094.492,-110.060,451.359,175.058,14.991,152.215
C00734=1094.498,-109.810,451.349,175.060,14.991,152.215
C00735=1094.504,-109.560,451.340,175.062,14.992,152.214
C00736=1094.510,-109.310,451.329,175.063,14.992,152.214
C00737=1094.516,-109.060,451.320,175.065,14.992,152.214
C00738=1094.522,-108.811,451.310,175.066,14.992,152.213
C00739=1094.528,-108.561,451.301,175.068,14.993,152.213
C00740=1094.535,-108.312,451.290,175.070,14.994,152.213
C00741=1094.541,-108.062,451.281,175.071,14.994,152.213
C00742=1094.547,-107.812,451.271,175.073,14.994,152.212
C00743=1094.553,-107.562,451.262,175.075,14.995,152.212
C00744=1094.559,-107.312,451.252,175.076,14.995,152.212
C00745=1094.565,-107.062,451.242,175.078,14.996,152.211
C00746=1094.571,-106.813,451.232,175.079,14.996,152.211
C00747=1094.577,-106.563,451.222,175.082,14.996,152.211
C00748=1094.584,-106.314,451.213,175.084,14.997,152.211
C00749=1094.589,-106.063,451.202,175.085,14.997,152.210
C00750=1094.595,-105.814,451.193,175.087,14.997,152.210
C00751=1094.602,-105.564,451.183,175.088,14.998,152.210
C00752=1094.608,-105.315,451.173,175.090,14.998,152.210
C00753=1094.614,-105.065,451.163,175.091,14.999,152.209
C00754=1094.619,-104.815,451.153,175.093,14.999,152.209
C00755=1094.626,-104.565,451.144,175.095,14.999,152.209
C00756=1094.632,-104.316,451.133,175.097,15.000,152.208
C00757=1094.638,-104.066,451.124,175.098,15.000,152.208
C00758=1094.644,-103.816,451.114,175.100,15.001,152.208
C00759=1094.650,-103.566,451.104,175.102,15.001,152.208
C00760=1094.656,-103.317,451.094,175.103,15.001,152.207
C00761=1094.663,-103.067,451.084,175.105,15.002,152.207
C00762=1094.668,-102.817,451.074,175.107,15.002,152.207
C00763=1094.674,-102.568,451.064,175.108,15.003,152.206
C00764=1094.681,-102.318,451.054,175.110,15.003,152.206
C00765=1094.687,-102.068,451.045,175.111,15.003,152.206
C00766=1094.692,-101.818,451.035,175.113,15.004,152.206
C00767=1094.699,-101.569,451.024,175.115,15.005,152.205
C00768=1094.705,-101.319,451.015,175.116,15.004,152.205
C00769=1094.710,-101.069,451.005,175.118,15.005,152.205
C00770=1094.717,-100.819,450.994,175.120,15.006,152.204
C00771=1094.724,-100.569,450.984,175.121,15.006,152.204
C00772=1094.730,-100.320,450.975,175.123,15.007,152.204
C00773=1094.735,-100.070,450.964,175.125,15.007,152.204
C00774=1094.742,-99.820,450.954,175.126,15.007,152.204
C00775=1094.748,-99.570,450.945,175.128,15.008,152.203
C00776=1094.754,-99.321,450.934,175.130,15.008,152.203
C00777=1094.760,-99.071,450.924,175.131,15.008,152.203
C00778=1094.766,-98.821,450.915,175.133,15.009,152.202
C00779=1094.772,-98.572,450.904,175.135,15.010,152.202
C00780=1094.778,-98.322,450.894,175.136,15.010,152.202
C00781=1094.784,-98.073,450.884,175.138,15.011,152.202
C00782=1094.790,-97.823,450.874,175.140,15.011,152.201
C00783=1094.796,-97.573,450.864,175.141,15.011,152.201
C00784=1094.802,-97.324,450.854,175.143,15.012,152.201
C00785=1094.809,-97.049,450.842,175.145,15.013,152.201
C00786=1094.816,-96.775,450.831,175.147,15.013,152.200
C00787=1094.822,-96.501,450.820,175.149,15.014,152.200
C00788=1094.828,-96.227,450.809,175.151,15.014,152.200
C00789=1094.835,-95.977,450.799,175.152,15.014,152.199
C00790=1094.840,-95.727,450.789,175.154,15.015,152.199
C00791=1094.847,-95.478,450.779,175.155,15.016,152.199
C00792=1094.852,-95.228,450.769,175.157,15.016,152.199
C00793=1094.858,-94.978,450.758,175.158,15.017,152.198
C00794=1094.864,-94.728,450.748,175.160,15.017,152.198
C00795=1094.870,-94.479,450.738,175.161,15.017,152.198
C00796=1094.876,-94.228,450.727,175.163,15.018,152.198
C00797=1094.883,-93.979,450.717,175.165,15.019,152.197
C00798=1094.888,-93.729,450.707,175.167,15.020,152.197
C00799=1094.895,-93.480,450.697,175.168,15.020,152.197
C00800=1094.900,-93.230,450.686,175.170,15.020,152.197
C00801=1094.907,-92.981,450.676,175.172,15.021,152.196
C00802=1094.912,-92.730,450.666,175.173,15.021,152.196
C00803=1094.919,-92.481,450.656,175.175,15.022,152.196
C00804=1094.924,-92.231,450.646,175.177,15.023,152.196
C00805=1094.931,-91.982,450.635,175.178,15.023,152.195
C00806=1094.936,-91.732,450.625,175.180,15.023,152.195
C00807=1094.943,-91.482,450.614,175.182,15.024,152.195
C00808=1094.948,-91.232,450.604,175.184,15.025,152.194
C00809=1094.955,-90.983,450.594,175.185,15.025,152.194
C00810=1094.960,-90.733,450.584,175.187,15.026,152.194
C00811=1094.966,-90.483,450.573,175.189,15.026,152.194
C00812=1094.973,-90.234,450.563,175.190,15.027,152.193
C00813=1094.978,-89.984,450.553,175.192,15.027,152.193
C00814=1094.985,-89.735,450.542,175.193,15.028,152.193
C00815=1094.991,-89.484,450.532,175.195,15.028,152.193
C00816=1094.997,-89.235,450.521,175.196,15.029,152.192
C00817=1095.003,-88.985,450.511,175.198,15.029,152.192
C00818=1095.009,-88.735,450.501,175.200,15.030,152.192
C00819=1095.015,-88.486,450.490,175.202,15.031,152.192
C00820=1095.020,-88.236,450.480,175.203,15.031,152.191
C00821=1095.027,-87.986,450.469,175.205,15.031,152.191
C00822=1095.033,-87.736,450.458,175.207,15.032,152.191
C00823=1095.039,-87.487,450.449,175.209,15.033,152.191
C00824=1095.045,-87.237,450.438,175.210,15.033,152.190
C00825=1095.051,-86.988,450.428,175.212,15.034,152.190
C00826=1095.057,-86.738,450.418,175.214,15.034,152.190
C00827=1095.063,-86.488,450.406,175.216,15.035,152.190
C00828=1095.070,-86.238,450.396,175.217,15.035,152.189
C00829=1095.075,-85.988,450.386,175.219,15.036,152.189
C00830=1095.081,-85.739,450.376,175.221,15.037,152.189
C00831=1095.087,-85.490,450.365,175.222,15.037,152.189
C00832=1095.093,-85.239,450.354,175.224,15.037,152.188
C00833=1095.100,-84.990,450.344,175.225,15.038,152.188
C00834=1095.105,-84.740,450.333,175.227,15.039,152.188
C00835=1095.111,-84.490,450.323,175.229,15.039,152.188
C00836=1095.118,-84.240,450.312,175.230,15.040,152.187
C00837=1095.124,-83.991,450.301,175.232,15.040,152.187
C00838=1095.130,-83.742,450.291,175.234,15.041,152.187
C00839=1095.136,-83.491,450.281,175.236,15.042,152.187
C00840=1095.141,-83.242,450.270,175.237,15.042,152.187
C00841=1095.148,-82.992,450.259,175.239,15.043,152.186
C00842=1095.154,-82.743,450.248,175.241,15.044,152.186
C00843=1095.160,-82.492,450.238,175.242,15.044,152.186
C00844=1095.166,-82.243,450.228,175.244,15.044,152.185
C00845=1095.172,-81.993,450.217,175.245,15.045,152.185
C00846=1095.179,-81.744,450.207,175.247,15.046,152.185
C00847=1095.184,-81.494,450.196,175.249,15.047,152.185
C00848=1095.191,-81.244,450.185,175.250,15.047,152.184
C00849=1095.197,-80.972,450.174,175.252,15.047,152.184
C00850=1095.204,-80.701,450.162,175.254,15.048,152.184
C00851=1095.211,-80.428,450.151,175.256,15.049,152.184
C00852=1095.218,-80.156,450.139,175.258,15.049,152.183
C00853=1095.223,-79.907,450.128,175.260,15.050,152.183
C00854=1095.229,-79.657,450.117,175.262,15.051,152.183
C00855=1095.235,-79.408,450.107,175.264,15.052,152.183
C00856=1095.241,-79.158,450.097,175.265,15.052,152.182
C00857=1095.247,-78.908,450.085,175.267,15.052,152.182
C00858=1095.253,-78.658,450.075,175.268,15.053,152.182
C00859=1095.259,-78.409,450.064,175.270,15.054,152.182
C00860=1095.264,-78.159,450.053,175.271,15.054,152.182
C00861=1095.272,-77.909,450.042,175.273,15.055,152.181
C00862=1095.277,-77.660,450.031,175.275,15.056,152.181
C00863=1095.283,-77.410,450.020,175.277,15.057,152.181
C00864=1095.288,-77.160,450.010,175.279,15.057,152.180
C00865=1095.295,-76.910,449.999,175.280,15.057,152.180
C00866=1095.301,-76.661,449.988,175.282,15.058,152.180
C00867=1095.307,-76.411,449.978,175.284,15.059,152.180
C00868=1095.313,-76.162,449.967,175.285,15.060,152.180
C00869=1095.319,-75.912,449.956,175.287,15.061,152.179
C00870=1095.325,-75.662,449.945,175.289,15.061,152.179
C00871=1095.331,-75.413,449.934,175.290,15.061,152.179
C00872=1095.337,-75.163,449.923,175.292,15.062,152.179
C00873=1095.343,-74.913,449.912,175.294,15.063,152.178
C00874=1095.349,-74.664,449.902,175.296,15.064,152.178
C00875=1095.355,-74.414,449.890,175.298,15.064,152.178
C00876=1095.361,-74.164,449.879,175.298,15.065,152.178
C00877=1095.367,-73.914,449.869,175.300,15.066,152.177
C00878=1095.372,-73.665,449.858,175.302,15.066,152.177
C00879=1095.379,-73.414,449.847,175.304,15.067,152.177
C00880=1095.384,-73.165,449.836,175.306,15.068,152.177
C00881=1095.390,-72.915,449.825,175.307,15.069,152.177
C00882=1095.396,-72.666,449.815,175.309,15.069,152.176
C00883=1095.402,-72.416,449.803,175.310,15.070,152.176
C00884=1095.408,-72.166,449.792,175.312,15.070,152.176
C00885=1095.414,-71.917,449.782,175.314,15.071,152.176
C00886=1095.420,-71.667,449.771,175.316,15.072,152.175
C00887=1095.426,-71.417,449.759,175.318,15.073,152.175
C00888=1095.431,-71.167,449.748,175.319,15.073,152.175
C00889=1095.437,-70.918,449.737,175.321,15.074,152.175
C00890=1095.442,-70.668,449.726,175.323,15.074,152.174
C00891=1095.449,-70.419,449.714,175.324,15.076,152.174
C00892=1095.455,-70.169,449.703,175.326,15.076,152.174
C00893=1095.460,-69.920,449.692,175.328,15.077,152.174
C00894=1095.467,-69.670,449.681,175.329,15.077,152.174
C00895=1095.473,-69.420,449.670,175.331,15.078,152.173
C00896=1095.478,-69.171,449.659,175.332,15.079,152.173
C00897=1095.485,-68.920,449.648,175.334,15.080,152.173
C00898=1095.490,-68.671,449.637,175.336,15.081,152.173
C00899=1095.496,-68.421,449.626,175.338,15.081,152.172
C00900=1095.502,-68.172,449.616,175.340,15.082,152.172
C00901=1095.508,-67.922,449.604,175.341,15.083,152.172
C00902=1095.513,-67.672,449.593,175.343,15.083,152.172
C00903=1095.519,-67.423,449.581,175.345,15.084,152.172
C00904=1095.526,-67.173,449.570,175.346,15.085,152.171
C00905=1095.531,-66.923,449.559,175.348,15.086,152.171
C00906=1095.538,-66.673,449.548,175.350,15.087,152.171
C00907=1095.543,-66.424,449.537,175.352,15.087,152.171
C00908=1095.549,-66.174,449.526,175.354,15.088,152.170
C00909=1095.555,-65.924,449.515,175.354,15.089,152.170
C00910=1095.562,-65.675,449.503,175.356,15.089,152.170
C00911=1095.567,-65.425,449.492,175.358,15.090,152.170
C00912=1095.573,-65.175,449.481,175.360,15.091,152.170
C00913=1095.579,-64.906,449.469,175.362,15.091,152.169
C00914=1095.586,-64.636,449.457,175.364,15.093,152.169
C00915=1095.591,-64.366,449.445,175.366,15.093,152.169
C00916=1095.599,-64.097,449.432,175.367,15.094,152.169
C00917=1095.605,-63.847,449.421,175.369,15.095,152.168
C00918=1095.610,-63.597,449.409,175.371,15.095,152.168
C00919=1095.616,-63.347,449.399,175.373,15.096,152.168
C00920=1095.622,-63.098,449.387,175.375,15.097,152.168
C00921=1095.628,-62.848,449.376,175.376,15.097,152.168
C00922=1095.634,-62.599,449.365,175.378,15.098,152.167
C00923=1095.641,-62.349,449.354,175.380,15.099,152.167
C00924=1095.646,-62.099,449.341,175.381,15.100,152.167
C00925=1095.652,-61.850,449.331,175.383,15.101,152.167
C00926=1095.658,-61.600,449.319,175.385,15.101,152.166
C00927=1095.664,-61.351,449.308,175.387,15.102,152.166
C00928=1095.670,-61.101,449.296,175.389,15.103,152.166
C00929=1095.676,-60.851,449.286,175.390,15.104,152.166
C00930=1095.682,-60.601,449.274,175.392,15.105,152.166
C00931=1095.688,-60.352,449.262,175.393,15.105,152.165
C00932=1095.693,-60.102,449.251,175.395,15.106,152.165
C00933=1095.700,-59.852,449.240,175.397,15.106,152.165
C00934=1095.706,-59.603,449.228,175.399,15.107,152.165
C00935=1095.711,-59.353,449.217,175.400,15.108,152.164
C00936=1095.717,-59.103,449.206,175.402,15.109,152.164
C00937=1095.724,-58.854,449.194,175.404,15.110,152.164
C00938=1095.730,-58.604,449.183,175.406,15.111,152.164
C00939=1095.736,-58.354,449.172,175.408,15.112,152.164
C00940=1095.741,-58.105,449.159,175.410,15.112,152.163
C00941=1095.748,-57.855,449.148,175.411,15.112,152.163
C00942=1095.754,-57.606,449.137,175.413,15.113,152.163
C00943=1095.760,-57.355,449.125,175.414,15.114,152.163
C00944=1095.766,-57.106,449.115,175.416,15.115,152.162
C00945=1095.772,-56.856,449.102,175.418,15.116,152.162
C00946=1095.777,-56.607,449.091,175.420,15.116,152.162
C00947=1095.784,-56.357,449.079,175.422,15.117,152.162
C00948=1095.790,-56.108,449.068,175.423,15.118,152.162
C00949=1095.796,-55.858,449.056,175.425,15.119,152.161
C00950=1095.801,-55.608,449.045,175.427,15.120,152.161
C00951=1095.808,-55.358,449.034,175.429,15.120,152.161
C00952=1095.814,-55.109,449.022,175.431,15.121,152.160
C00953=1095.819,-54.859,449.010,175.432,15.122,152.160
C00954=1095.825,-54.610,448.999,175.433,15.122,152.160
C00955=1095.832,-54.360,448.987,175.435,15.123,152.160
C00956=1095.838,-54.110,448.975,175.437,15.124,152.160
C00957=1095.843,-53.860,448.964,175.439,15.125,152.160
C00958=1095.850,-53.611,448.952,175.441,15.126,152.159
C00959=1095.856,-53.361,448.941,175.443,15.126,152.159
C00960=1095.862,-53.111,448.928,175.444,15.127,152.159
C00961=1095.867,-52.862,448.918,175.446,15.128,152.158
C00962=1095.874,-52.612,448.906,175.448,15.129,152.158
C00963=1095.880,-52.362,448.894,175.450,15.130,152.158
C00964=1095.886,-52.113,448.882,175.452,15.130,152.158
C00965=1095.892,-51.863,448.870,175.454,15.131,152.158
C00966=1095.898,-51.614,448.859,175.455,15.132,152.157
C00967=1095.904,-51.364,448.847,175.456,15.133,152.157
C00968=1095.910,-51.114,448.836,175.458,15.133,152.157
C00969=1095.916,-50.865,448.824,175.460,15.134,152.157
C00970=1095.922,-50.614,448.812,175.462,15.135,152.156
C00971=1095.928,-50.365,448.801,175.464,15.135,152.156
C00972=1095.934,-50.116,448.788,175.465,15.137,152.156
C00973=1095.940,-49.866,448.777,175.467,15.137,152.156
C00974=1095.946,-49.616,448.765,175.469,15.138,152.156
C00975=1095.951,-49.367,448.754,175.471,15.139,152.155
C00976=1095.957,-49.117,448.741,175.473,15.140,152.155
C00977=1095.964,-48.849,448.729,175.475,15.141,152.155
C00978=1095.970,-48.580,448.716,175.476,15.141,152.155
C00979=1095.976,-48.312,448.703,175.478,15.142,152.155
C00980=1095.983,-48.043,448.691,175.481,15.144,152.154
C00981=1095.988,-47.794,448.679,175.482,15.144,152.154
C00982=1095.995,-47.544,448.667,175.484,15.145,152.154
C00983=1096.000,-47.294,448.655,175.485,15.146,152.154
C00984=1096.006,-47.045,448.643,175.487,15.147,152.153
C00985=1096.012,-46.795,448.631,175.489,15.147,152.153
C00986=1096.017,-46.545,448.619,175.491,15.148,152.153
C00987=1096.024,-46.296,448.607,175.492,15.149,152.153
C00988=1096.029,-46.046,448.595,175.494,15.150,152.153
C00989=1096.036,-45.796,448.584,175.496,15.151,152.152
C00990=1096.041,-45.547,448.572,175.498,15.152,152.152
C00991=1096.048,-45.298,448.560,175.500,15.152,152.152
C00992=1096.053,-45.048,448.547,175.502,15.153,152.152
C00993=1096.058,-44.798,448.536,175.503,15.154,152.152
C00994=1096.065,-44.548,448.524,175.505,15.155,152.151
C00995=1096.070,-44.299,448.512,175.507,15.156,152.151
C00996=1096.077,-44.049,448.500,175.508,15.157,152.151
C00997=1096.083,-43.799,448.488,175.510,15.158,152.151
C00998=1096.089,-43.550,448.476,175.512,15.158,152.150
C00999=1096.095,-43.300,448.464,175.514,15.159,152.150
C01000=1096.101,-43.050,448.451,175.516,15.160,152.150
C01001=1096.106,-42.801,448.440,175.518,15.161,152.150
C01002=1096.112,-42.551,448.428,175.519,15.162,152.150
C01003=1096.118,-42.302,448.416,175.521,15.162,152.149
C01004=1096.124,-42.052,448.404,175.523,15.164,152.149
C01005=1096.130,-41.802,448.392,175.525,15.164,152.149
C01006=1096.136,-41.553,448.380,175.527,15.165,152.149
C01007=1096.142,-41.303,448.368,175.528,15.166,152.149
C01008=1096.148,-41.053,448.355,175.530,15.167,152.148
C01009=1096.154,-40.804,448.343,175.532,15.168,152.148
C01010=1096.160,-40.554,448.331,175.534,15.168,152.148
C01011=1096.166,-40.304,448.320,175.536,15.170,152.148
C01012=1096.171,-40.055,448.307,175.537,15.170,152.147
C01013=1096.177,-39.805,448.295,175.539,15.171,152.147
C01014=1096.184,-39.556,448.283,175.541,15.172,152.147
C01015=1096.190,-39.306,448.270,175.543,15.173,152.147
C01016=1096.195,-39.056,448.258,175.545,15.174,152.147
C01017=1096.202,-38.807,448.246,175.547,15.174,152.146
C01018=1096.208,-38.557,448.234,175.548,15.175,152.146
C01019=1096.213,-38.308,448.221,175.550,15.176,152.146
C01020=1096.218,-38.057,448.210,175.552,15.177,152.146
C01021=1096.224,-37.807,448.197,175.554,15.178,152.145
C01022=1096.230,-37.559,448.185,175.555,15.179,152.145
C01023=1096.236,-37.309,448.173,175.557,15.180,152.145
C01024=1096.242,-37.059,448.161,175.559,15.180,152.145
C01025=1096.247,-36.810,448.148,175.561,15.182,152.145
C01026=1096.253,-36.560,448.136,175.563,15.182,152.144
C01027=1096.260,-36.310,448.124,175.564,15.183,152.144
C01028=1096.265,-36.061,448.111,175.566,15.184,152.144
C01029=1096.271,-35.811,448.099,175.568,15.185,152.144
C01030=1096.277,-35.561,448.086,175.570,15.186,152.144
C01031=1096.282,-35.312,448.074,175.571,15.187,152.143
C01032=1096.288,-35.062,448.062,175.573,15.188,152.143
C01033=1096.295,-34.813,448.050,175.575,15.188,152.143
C01034=1096.300,-34.563,448.037,175.578,15.190,152.143
C01035=1096.306,-34.314,448.025,175.579,15.191,152.143
C01036=1096.312,-34.064,448.012,175.581,15.191,152.142
C01037=1096.318,-33.814,448.000,175.583,15.192,152.142
C01038=1096.323,-33.565,447.988,175.585,15.193,152.142
C01039=1096.330,-33.315,447.976,175.587,15.194,152.142
C01040=1096.336,-33.065,447.963,175.588,15.195,152.141
C01041=1096.342,-32.797,447.950,175.590,15.196,152.141
C01042=1096.349,-32.529,447.936,175.592,15.197,152.141
C01043=1096.354,-32.261,447.923,175.594,15.197,152.141
C01044=1096.361,-31.993,447.910,175.597,15.199,152.140
C01045=1096.366,-31.743,447.897,175.598,15.199,152.140
C01046=1096.372,-31.493,447.885,175.600,15.201,152.140
C01047=1096.378,-31.244,447.872,175.602,15.201,152.140
C01048=1096.384,-30.994,447.860,175.604,15.202,152.140
C01049=1096.390,-30.745,447.847,175.605,15.203,152.139
C01050=1096.396,-30.496,447.835,175.607,15.204,152.139
C01051=1096.402,-30.246,447.822,175.609,15.205,152.139
C01052=1096.408,-29.996,447.810,175.611,15.205,152.139
C01053=1096.413,-29.747,447.798,175.613,15.207,152.139
C01054=1096.419,-29.497,447.785,175.614,15.207,152.138
C01055=1096.425,-29.247,447.772,175.616,15.208,152.138
C01056=1096.431,-28.998,447.759,175.618,15.209,152.138
C01057=1096.437,-28.748,447.747,175.620,15.210,152.138
C01058=1096.443,-28.499,447.734,175.622,15.211,152.137
C01059=1096.449,-28.249,447.722,175.624,15.211,152.137
C01060=1096.455,-27.999,447.710,175.625,15.213,152.137
C01061=1096.461,-27.750,447.697,175.627,15.213,152.137
C01062=1096.467,-27.500,447.684,175.629,15.214,152.137
C01063=1096.473,-27.250,447.672,175.632,15.215,152.136
C01064=1096.478,-27.001,447.659,175.633,15.217,152.136
C01065=1096.484,-26.751,447.647,175.635,15.217,152.136
C01066=1096.491,-26.502,447.634,175.637,15.218,152.136
C01067=1096.497,-26.252,447.621,175.639,15.219,152.135
C01068=1096.502,-26.002,447.608,175.640,15.220,152.135
C01069=1096.507,-25.752,447.596,175.642,15.221,152.135
C01070=1096.513,-25.503,447.582,175.644,15.221,152.135
C01071=1096.519,-25.253,447.570,175.646,15.223,152.135
C01072=1096.525,-25.003,447.557,175.648,15.223,152.134
C01073=1096.531,-24.754,447.545,175.649,15.224,152.134
C01074=1096.537,-24.505,447.532,175.651,15.225,152.134
C01075=1096.542,-24.255,447.519,175.653,15.226,152.134
C01076=1096.548,-24.005,447.507,175.656,15.227,152.134
C01077=1096.555,-23.756,447.493,175.657,15.228,152.133
C01078=1096.560,-23.506,447.480,175.659,15.229,152.133
C01079=1096.565,-23.257,447.468,175.661,15.230,152.133
C01080=1096.571,-23.007,447.456,175.663,15.231,152.133
C01081=1096.577,-22.757,447.442,175.664,15.232,152.133
C01082=1096.583,-22.508,447.430,175.666,15.232,152.132
C01083=1096.589,-22.258,447.416,175.668,15.233,152.132
C01084=1096.595,-22.008,447.404,175.670,15.234,152.132
C01085=1096.601,-21.759,447.391,175.672,15.235,152.132
C01086=1096.606,-21.510,447.378,175.673,15.236,152.131
C01087=1096.612,-21.260,447.365,175.676,15.237,152.131
C01088=1096.618,-21.010,447.353,175.678,15.238,152.131
C01089=1096.624,-20.761,447.339,175.680,15.239,152.131
C01090=1096.630,-20.511,447.327,175.682,15.240,152.131
C01091=1096.636,-20.261,447.314,175.683,15.240,152.130
C01092=1096.641,-20.011,447.301,175.685,15.242,152.130
C01093=1096.647,-19.761,447.288,175.687,15.242,152.130
C01094=1096.653,-19.513,447.275,175.689,15.243,152.130
C01095=1096.659,-19.263,447.263,175.691,15.244,152.129
C01096=1096.665,-19.014,447.249,175.692,15.245,152.129
C01097=1096.671,-18.764,447.237,175.695,15.246,152.129
C01098=1096.676,-18.514,447.223,175.697,15.247,152.129
C01099=1096.682,-18.264,447.210,175.699,15.248,152.128
C01100=1096.688,-18.015,447.197,175.700,15.249,152.128
C01101=1096.694,-17.765,447.184,175.702,15.250,152.128
C01102=1096.701,-17.516,447.171,175.704,15.250,152.128
C01103=1096.706,-17.266,447.158,175.706,15.251,152.128
C01104=1096.712,-17.016,447.145,175.707,15.252,152.128
C01105=1096.718,-16.748,447.131,175.710,15.254,152.127
C01106=1096.724,-16.479,447.117,175.712,15.254,152.127
C01107=1096.731,-16.209,447.103,175.714,15.255,152.127
C01108=1096.737,-15.941,447.089,175.716,15.256,152.126
C01109=1096.743,-15.691,447.076,175.718,15.257,152.126
C01110=1096.749,-15.442,447.063,175.720,15.258,152.126
C01111=1096.755,-15.192,447.050,175.722,15.259,152.126
C01112=1096.761,-14.943,447.037,175.724,15.260,152.126
C01113=1096.766,-14.693,447.023,175.726,15.260,152.125
C01114=1096.772,-14.443,447.010,175.727,15.262,152.125
C01115=1096.778,-14.194,446.997,175.729,15.262,152.125
C01116=1096.783,-13.944,446.984,175.731,15.263,152.125
C01117=1096.789,-13.695,446.971,175.733,15.265,152.125
C01118=1096.795,-13.445,446.958,175.735,15.266,152.124
C01119=1096.801,-13.196,446.945,175.737,15.266,152.124
C01120=1096.807,-12.946,446.931,175.739,15.267,152.124
C01121=1096.812,-12.696,446.918,175.741,15.268,152.124
C01122=1096.818,-12.447,446.905,175.742,15.269,152.123
C01123=1096.824,-12.198,446.892,175.744,15.270,152.123
C01124=1096.830,-11.947,446.878,175.747,15.271,152.123
C01125=1096.836,-11.698,446.865,175.749,15.272,152.123
C01126=1096.841,-11.448,446.852,175.750,15.273,152.122
C01127=1096.847,-11.199,446.839,175.752,15.274,152.122
C01128=1096.853,-10.949,446.825,175.754,15.274,152.122
C01129=1096.859,-10.700,446.812,175.756,15.276,152.122
C01130=1096.865,-10.450,446.799,175.758,15.276,152.122
C01131=1096.870,-10.200,446.785,175.760,15.278,152.121
C01132=1096.876,-9.951,446.772,175.762,15.278,152.121
C01133=1096.882,-9.701,446.759,175.764,15.279,152.121
C01134=1096.888,-9.452,446.746,175.766,15.280,152.121
C01135=1096.894,-9.202,446.732,175.768,15.281,152.120
C01136=1096.900,-8.953,446.718,175.769,15.282,152.120
C01137=1096.905,-8.703,446.706,175.771,15.282,152.120
C01138=1096.911,-8.453,446.692,175.774,15.284,152.120
C01139=1096.917,-8.204,446.679,175.776,15.285,152.120
C01140=1096.923,-7.955,446.665,175.777,15.286,152.119
C01141=1096.929,-7.705,446.652,175.779,15.286,152.119
C01142=1096.934,-7.455,446.638,175.781,15.287,152.119
C01143=1096.940,-7.206,446.625,175.783,15.288,152.119
C01144=1096.946,-6.956,446.611,175.785,15.289,152.118
C01145=1096.952,-6.706,446.599,175.787,15.290,152.118
C01146=1096.957,-6.457,446.585,175.789,15.291,152.118
C01147=1096.964,-6.207,446.571,175.791,15.292,152.118
C01148=1096.969,-5.957,446.557,175.793,15.293,152.117
C01149=1096.976,-5.708,446.544,175.795,15.293,152.117
C01150=1096.981,-5.458,446.530,175.796,15.294,152.117
C01151=1096.987,-5.209,446.518,175.799,15.296,152.117
C01152=1096.992,-4.959,446.504,175.801,15.297,152.116
C01153=1096.999,-4.710,446.491,175.803,15.297,152.116
C01154=1097.004,-4.460,446.477,175.805,15.298,152.116
C01155=1097.010,-4.211,446.463,175.807,15.299,152.116
C01156=1097.016,-3.961,446.450,175.808,15.300,152.116
C01157=1097.022,-3.712,446.436,175.811,15.301,152.115
C01158=1097.028,-3.462,446.422,175.813,15.302,152.115
C01159=1097.034,-3.213,446.409,175.815,15.303,152.115
C01160=1097.039,-2.962,446.396,175.817,15.303,152.115
C01161=1097.045,-2.713,446.382,175.818,15.305,152.114
C01162=1097.051,-2.463,446.368,175.820,15.305,152.114
C01163=1097.057,-2.214,446.355,175.823,15.307,152.114
C01164=1097.062,-1.964,446.341,175.825,15.307,152.114
C01165=1097.068,-1.715,446.327,175.826,15.308,152.113
C01166=1097.074,-1.465,446.314,175.828,15.309,152.113
C01167=1097.079,-1.216,446.300,175.830,15.310,152.113
C01168=1097.085,-0.966,446.286,175.833,15.311,152.113
C01169=1097.092,-0.696,446.271,175.834,15.312,152.112
C01170=1097.098,-0.425,446.256,175.836,15.313,152.112
C01171=1097.103,-0.155,446.242,175.839,15.314,152.112
C01172=1097.110,0.116,446.227,175.841,15.315,152.112
C01173=1097.116,0.365,446.213,175.842,15.316,152.112
C01174=1097.121,0.615,446.199,175.844,15.317,152.111
C01175=1097.127,0.864,446.185,175.847,15.318,152.111
C01176=1097.133,1.114,446.172,175.849,15.319,152.111
C01177=1097.138,1.363,446.158,175.851,15.319,152.111
C01178=1097.144,1.614,446.144,175.852,15.321,152.110
C01179=1097.150,1.863,446.130,175.854,15.321,152.110
C01180=1097.156,2.112,446.116,175.857,15.323,152.110
C01181=1097.162,2.361,446.102,175.859,15.323,152.110
C01182=1097.167,2.611,446.088,175.861,15.324,152.109
C01183=1097.173,2.861,446.075,175.863,15.325,152.109
C01184=1097.178,3.110,446.061,175.864,15.326,152.109
C01185=1097.185,3.360,446.047,175.867,15.327,152.109
C01186=1097.191,3.610,446.033,175.869,15.328,152.108
C01187=1097.196,3.859,446.019,175.871,15.329,152.108
C01188=1097.201,4.109,446.005,175.872,15.330,152.108
C01189=1097.207,4.358,445.992,175.874,15.330,152.108
C01190=1097.213,4.607,445.978,175.877,15.332,152.107
C01191=1097.220,4.857,445.963,175.879,15.332,152.107
C01192=1097.225,5.107,445.949,175.881,15.333,152.107
C01193=1097.230,5.356,445.936,175.882,15.334,152.107
C01194=1097.236,5.606,445.922,175.884,15.335,152.107
C01195=1097.242,5.855,445.908,175.887,15.336,152.106
C01196=1097.249,6.105,445.894,175.889,15.337,152.106
C01197=1097.254,6.355,445.880,175.891,15.338,152.106
C01198=1097.260,6.604,445.866,175.893,15.338,152.105
C01199=1097.265,6.854,445.852,175.894,15.339,152.105
C01200=1097.270,7.103,445.838,175.897,15.341,152.105
C01201=1097.278,7.353,445.824,175.899,15.341,152.105
C01202=1097.283,7.602,445.810,175.901,15.342,152.104
C01203=1097.289,7.852,445.796,175.903,15.343,152.104
C01204=1097.294,8.101,445.782,175.905,15.344,152.104
C01205=1097.300,8.351,445.767,175.907,15.345,152.104
C01206=1097.306,8.601,445.753,175.909,15.346,152.104
C01207=1097.311,8.850,445.739,175.911,15.347,152.103
C01208=1097.317,9.100,445.726,175.913,15.347,152.103
C01209=1097.324,9.349,445.711,175.915,15.349,152.103
C01210=1097.329,9.599,445.697,175.917,15.349,152.102
C01211=1097.335,9.848,445.684,175.919,15.350,152.102
C01212=1097.341,10.097,445.669,175.921,15.351,152.102
C01213=1097.347,10.347,445.655,175.923,15.352,152.102
C01214=1097.352,10.597,445.641,175.925,15.353,152.101
C01215=1097.358,10.846,445.626,175.927,15.354,152.101
C01216=1097.364,11.096,445.612,175.929,15.354,152.101
C01217=1097.370,11.346,445.598,175.931,15.355,152.101
C01218=1097.376,11.594,445.584,175.934,15.356,152.100
C01219=1097.382,11.844,445.570,175.936,15.357,152.100
C01220=1097.388,12.094,445.555,175.938,15.358,152.100
C01221=1097.393,12.343,445.541,175.939,15.359,152.100
C01222=1097.399,12.593,445.528,175.941,15.359,152.099
C01223=1097.405,12.843,445.513,175.944,15.361,152.099
C01224=1097.411,13.092,445.499,175.946,15.361,152.099
C01225=1097.417,13.341,445.484,175.948,15.362,152.099
C01226=1097.423,13.591,445.470,175.950,15.363,152.098
C01227=1097.428,13.841,445.456,175.952,15.364,152.098
C01228=1097.434,14.090,445.442,175.954,15.365,152.098
C01229=1097.440,14.340,445.427,175.956,15.366,152.098
C01230=1097.446,14.589,445.413,175.958,15.366,152.097
C01231=1097.451,14.839,445.399,175.961,15.368,152.097
C01232=1097.458,15.088,445.384,175.962,15.368,152.097
C01233=1097.463,15.361,445.368,175.964,15.369,152.096
C01234=1097.470,15.633,445.353,175.967,15.370,152.096
C01235=1097.476,15.906,445.338,175.969,15.371,152.096
C01236=1097.483,16.179,445.322,175.972,15.372,152.095
C01237=1097.488,16.428,445.307,175.974,15.373,152.095
C01238=1097.494,16.677,445.293,175.976,15.373,152.095
C01239=1097.500,16.927,445.278,175.978,15.374,152.095
C01240=1097.506,17.176,445.264,175.980,15.376,152.094
C01241=1097.511,17.426,445.249,175.982,15.376,152.094
C01242=1097.517,17.676,445.234,175.984,15.377,152.094
C01243=1097.523,17.925,445.220,175.986,15.378,152.094
C01244=1097.528,18.174,445.206,175.989,15.379,152.093
C01245=1097.534,18.424,445.192,175.990,15.380,152.093
C01246=1097.540,18.673,445.177,175.992,15.381,152.093
C01247=1097.546,18.923,445.163,175.994,15.381,152.093
C01248=1097.552,19.173,445.148,175.997,15.383,152.092
C01249=1097.557,19.422,445.133,175.999,15.383,152.092
C01250=1097.563,19.671,445.119,176.001,15.384,152.092
C01251=1097.569,19.921,445.104,176.002,15.385,152.092
C01252=1097.575,20.170,445.090,176.005,15.386,152.091
C01253=1097.581,20.420,445.075,176.007,15.387,152.091
C01254=1097.586,20.670,445.060,176.009,15.387,152.091
C01255=1097.591,20.919,445.046,176.012,15.388,152.090
C01256=1097.598,21.169,445.031,176.014,15.389,152.090
C01257=1097.603,21.418,445.017,176.016,15.390,152.090
C01258=1097.609,21.668,445.002,176.018,15.391,152.090
C01259=1097.615,21.917,444.987,176.020,15.392,152.089
C01260=1097.620,22.166,444.973,176.022,15.393,152.089
C01261=1097.627,22.416,444.958,176.024,15.393,152.089
C01262=1097.632,22.666,444.943,176.026,15.394,152.088
C01263=1097.638,22.915,444.928,176.029,15.395,152.088
C01264=1097.644,23.164,444.914,176.030,15.396,152.088
C01265=1097.649,23.414,444.900,176.032,15.397,152.088
C01266=1097.655,23.664,444.884,176.034,15.398,152.087
C01267=1097.661,23.913,444.870,176.037,15.398,152.087
C01268=1097.667,24.163,444.855,176.039,15.399,152.087
C01269=1097.672,24.412,444.840,176.041,15.400,152.086
C01270=1097.678,24.662,444.826,176.044,15.401,152.086
C01271=1097.684,24.911,444.811,176.045,15.402,152.086
C01272=1097.690,25.160,444.796,176.047,15.403,152.086
C01273=1097.695,25.410,444.781,176.049,15.403,152.085
C01274=1097.701,25.660,444.767,176.052,15.404,152.085
C01275=1097.707,25.909,444.752,176.054,15.405,152.085
C01276=1097.712,26.158,444.737,176.056,15.406,152.084
C01277=1097.719,26.408,444.722,176.059,15.407,152.084
C01278=1097.724,26.657,444.707,176.060,15.408,152.084
C01279=1097.730,26.907,444.692,176.062,15.409,152.084
C01280=1097.735,27.157,444.678,176.065,15.409,152.083
C01281=1097.742,27.406,444.663,176.067,15.410,152.083
C01282=1097.747,27.656,444.648,176.069,15.411,152.083
C01283=1097.753,27.905,444.633,176.071,15.412,152.082
C01284=1097.758,28.154,444.618,176.074,15.413,152.082
C01285=1097.765,28.404,444.603,176.076,15.414,152.082
C01286=1097.771,28.653,444.588,176.078,15.414,152.082
C01287=1097.776,28.903,444.573,176.080,15.415,152.081
C01288=1097.782,29.152,444.558,176.082,15.416,152.081
C01289=1097.787,29.403,444.543,176.084,15.417,152.081
C01290=1097.793,29.652,444.529,176.086,15.417,152.080
C01291=1097.799,29.901,444.513,176.089,15.419,152.080
C01292=1097.804,30.150,444.498,176.091,15.419,152.080
C01293=1097.810,30.400,444.483,176.093,15.420,152.080
C01294=1097.816,30.649,444.468,176.095,15.421,152.079
C01295=1097.822,30.899,444.453,176.097,15.422,152.079
C01296=1097.827,31.148,444.438,176.099,15.422,152.079
C01297=1097.834,31.422,444.421,176.102,15.423,152.078
C01298=1097.840,31.696,444.404,176.104,15.424,152.078
C01299=1097.846,31.970,444.389,176.107,15.425,152.078
C01300=1097.852,32.244,444.372,176.109,15.426,152.077
C01301=1097.859,32.493,444.357,176.112,15.427,152.077
C01302=1097.864,32.743,444.342,176.113,15.428,152.077
C01303=1097.869,32.993,444.326,176.116,15.428,152.076
C01304=1097.875,33.241,444.311,176.118,15.429,152.076
C01305=1097.881,33.491,444.296,176.120,15.430,152.076
C01306=1097.887,33.740,444.281,176.122,15.431,152.076
C01307=1097.892,33.990,444.266,176.124,15.431,152.075
C01308=1097.899,34.240,444.251,176.127,15.432,152.075
C01309=1097.904,34.489,444.236,176.129,15.433,152.075
C01310=1097.910,34.739,444.221,176.131,15.434,152.074
C01311=1097.915,34.988,444.206,176.134,15.435,152.074
C01312=1097.922,35.237,444.190,176.136,15.435,152.074
C01313=1097.927,35.487,444.175,176.137,15.436,152.073
C01314=1097.932,35.737,444.159,176.140,15.437,152.073
C01315=1097.939,35.986,444.144,176.142,15.438,152.073
C01316=1097.944,36.235,444.129,176.144,15.438,152.072
C01317=1097.950,36.485,444.114,176.147,15.439,152.072
C01318=1097.956,36.735,444.099,176.149,15.440,152.072
C01319=1097.961,36.984,444.083,176.151,15.441,152.072
C01320=1097.968,37.233,444.068,176.154,15.442,152.071
C01321=1097.973,37.483,444.053,176.156,15.442,152.071
C01322=1097.979,37.732,444.038,176.158,15.443,152.071
C01323=1097.985,37.982,444.022,176.161,15.444,152.070
C01324=1097.990,38.231,444.006,176.162,15.445,152.070
C01325=1097.996,38.481,443.991,176.164,15.445,152.070
C01326=1098.002,38.730,443.976,176.167,15.446,152.069
C01327=1098.007,38.980,443.960,176.169,15.447,152.069
C01328=1098.013,39.229,443.944,176.171,15.448,152.069
C01329=1098.019,39.478,443.930,176.174,15.449,152.068
C01330=1098.025,39.728,443.914,176.176,15.449,152.068
C01331=1098.030,39.977,443.899,176.178,15.450,152.068
C01332=1098.036,40.227,443.883,176.181,15.451,152.067
C01333=1098.042,40.476,443.868,176.183,15.452,152.067
C01334=1098.047,40.726,443.853,176.185,15.452,152.067
C01335=1098.053,40.976,443.837,176.188,15.453,152.066
C01336=1098.059,41.225,443.821,176.189,15.454,152.066
C01337=1098.064,41.474,443.806,176.191,15.455,152.066
C01338=1098.070,41.724,443.791,176.194,15.456,152.065
C01339=1098.076,41.973,443.774,176.196,15.456,152.065
C01340=1098.081,42.222,443.759,176.198,15.457,152.065
C01341=1098.087,42.472,443.744,176.201,15.458,152.064
C01342=1098.093,42.721,443.728,176.203,15.459,152.064
C01343=1098.098,42.971,443.713,176.205,15.459,152.064
C01344=1098.104,43.220,443.697,176.208,15.460,152.064
C01345=1098.110,43.470,443.681,176.210,15.461,152.063
C01346=1098.116,43.719,443.666,176.212,15.461,152.063
C01347=1098.122,43.968,443.650,176.214,15.463,152.063
C01348=1098.127,44.218,443.635,176.217,15.463,152.062
C01349=1098.133,44.467,443.619,176.219,15.464,152.062
C01350=1098.138,44.717,443.603,176.222,15.464,152.061
C01351=1098.144,44.967,443.588,176.223,15.465,152.061
C01352=1098.149,45.216,443.572,176.225,15.466,152.061
C01353=1098.155,45.466,443.556,176.228,15.467,152.061
C01354=1098.161,45.715,443.540,176.230,15.468,152.060
C01355=1098.166,45.964,443.525,176.233,15.468,152.060
C01356=1098.172,46.213,443.509,176.235,15.469,152.060
C01357=1098.178,46.463,443.493,176.237,15.470,152.059
C01358=1098.183,46.712,443.477,176.240,15.471,152.059
C01359=1098.189,46.962,443.462,176.242,15.471,152.059
C01360=1098.194,47.211,443.445,176.244,15.472,152.058
C01361=1098.201,47.486,443.428,176.247,15.473,152.058
C01362=1098.207,47.760,443.412,176.250,15.474,152.057
C01363=1098.213,48.033,443.393,176.252,15.474,152.057
C01364=1098.219,48.307,443.376,176.254,15.476,152.057
C01365=1098.225,48.557,443.360,176.257,15.476,152.056
C01366=1098.230,48.806,443.345,176.259,15.477,152.056
C01367=1098.236,49.055,443.329,176.261,15.477,152.056
C01368=1098.242,49.305,443.313,176.263,15.478,152.055
C01369=1098.247,49.555,443.297,176.266,15.479,152.055
C01370=1098.253,49.803,443.281,176.268,15.480,152.055
C01371=1098.258,50.053,443.266,176.270,15.480,152.054
C01372=1098.264,50.303,443.249,176.273,15.481,152.054
C01373=1098.270,50.552,443.233,176.275,15.482,152.054
C01374=1098.275,50.801,443.218,176.277,15.482,152.053
C01375=1098.281,51.051,443.202,176.280,15.483,152.053
C01376=1098.287,51.300,443.185,176.282,15.484,152.053
C01377=1098.293,51.550,443.170,176.285,15.485,152.052
C01378=1098.298,51.799,443.154,176.287,15.486,152.052
C01379=1098.304,52.048,443.138,176.289,15.486,152.052
C01380=1098.310,52.298,443.122,176.292,15.487,152.051
C01381=1098.315,52.548,443.105,176.294,15.487,152.051
C01382=1098.321,52.797,443.089,176.296,15.488,152.050
C01383=1098.326,53.046,443.074,176.299,15.489,152.050
C01384=1098.332,53.296,443.058,176.301,15.489,152.050
C01385=1098.338,53.545,443.041,176.304,15.490,152.049
C01386=1098.344,53.794,443.025,176.306,15.491,152.049
C01387=1098.350,54.044,443.010,176.308,15.491,152.049
C01388=1098.356,54.294,442.993,176.311,15.492,152.048
C01389=1098.361,54.542,442.977,176.313,15.493,152.048
C01390=1098.367,54.792,442.961,176.316,15.494,152.048
C01391=1098.372,55.042,442.946,176.318,15.494,152.047
C01392=1098.378,55.291,442.929,176.320,15.495,152.047
C01393=1098.384,55.541,442.912,176.323,15.495,152.046
C01394=1098.390,55.790,442.896,176.325,15.496,152.046
C01395=1098.396,56.039,442.880,176.327,15.496,152.046
C01396=1098.401,56.289,442.865,176.330,15.497,152.045
C01397=1098.407,56.538,442.849,176.332,15.498,152.045
C01398=1098.412,56.787,442.832,176.335,15.499,152.045
C01399=1098.418,57.037,442.816,176.337,15.499,152.044
C01400=1098.424,57.286,442.799,176.339,15.499,152.044
C01401=1098.430,57.536,442.783,176.342,15.501,152.044
C01402=1098.436,57.785,442.767,176.344,15.501,152.043
C01403=1098.441,58.035,442.751,176.347,15.502,152.043
C01404=1098.447,58.284,442.735,176.349,15.502,152.042
C01405=1098.453,58.534,442.719,176.351,15.503,152.042
C01406=1098.458,58.783,442.702,176.354,15.504,152.042
C01407=1098.464,59.032,442.686,176.356,15.504,152.041
C01408=1098.470,59.281,442.670,176.358,15.504,152.041
C01409=1098.476,59.531,442.653,176.361,15.506,152.041
C01410=1098.482,59.780,442.637,176.363,15.506,152.040
C01411=1098.487,60.029,442.621,176.366,15.507,152.040
C01412=1098.493,60.279,442.604,176.368,15.507,152.039
C01413=1098.499,60.528,442.588,176.370,15.507,152.039
C01414=1098.505,60.778,442.571,176.373,15.509,152.039
C01415=1098.511,61.027,442.555,176.375,15.509,152.038
C01416=1098.516,61.277,442.538,176.378,15.510,152.038
C01417=1098.522,61.526,442.522,176.380,15.510,152.037
C01418=1098.528,61.775,442.506,176.383,15.510,152.037
C01419=1098.534,62.025,442.490,176.386,15.511,152.036
C01420=1098.540,62.274,442.473,176.388,15.512,152.036
C01421=1098.545,62.524,442.457,176.390,15.513,152.036
C01422=1098.551,62.773,442.440,176.393,15.513,152.035
C01423=1098.557,63.022,442.424,176.395,15.513,152.035
C01424=1098.563,63.272,442.408,176.398,15.514,152.034
C01425=1098.568,63.546,442.390,176.400,15.515,152.034
C01426=1098.575,63.820,442.372,176.403,15.515,152.034
C01427=1098.582,64.093,442.353,176.406,15.516,152.033
C01428=1098.588,64.366,442.335,176.408,15.517,152.033
C01429=1098.593,64.616,442.318,176.411,15.518,152.032
C01430=1098.599,64.865,442.302,176.413,15.518,152.032
C01431=1098.605,65.115,442.286,176.416,15.519,152.031
C01432=1098.610,65.364,442.269,176.418,15.519,152.031
C01433=1098.617,65.613,442.252,176.421,15.519,152.031
C01434=1098.622,65.863,442.235,176.424,15.520,152.030
C01435=1098.628,66.112,442.219,176.426,15.520,152.030
C01436=1098.634,66.361,442.203,176.428,15.522,152.030
C01437=1098.639,66.611,442.186,176.431,15.522,152.029
C01438=1098.645,66.860,442.169,176.434,15.523,152.029
C01439=1098.650,67.110,442.152,176.436,15.523,152.028
C01440=1098.656,67.359,442.136,176.438,15.523,152.028
C01441=1098.662,67.609,442.119,176.441,15.524,152.027
C01442=1098.668,67.858,442.102,176.443,15.525,152.027
C01443=1098.673,68.108,442.086,176.446,15.525,152.027
C01444=1098.679,68.356,442.069,176.448,15.526,152.026
C01445=1098.684,68.606,442.052,176.450,15.526,152.026
C01446=1098.690,68.855,442.036,176.453,15.527,152.025
C01447=1098.696,69.105,442.018,176.456,15.527,152.025
C01448=1098.702,69.354,442.001,176.459,15.528,152.024
C01449=1098.708,69.604,441.984,176.461,15.528,152.024
C01450=1098.713,69.853,441.968,176.464,15.529,152.024
C01451=1098.719,70.102,441.951,176.466,15.529,152.023
C01452=1098.725,70.352,441.934,176.468,15.530,152.023
C01453=1098.730,70.601,441.918,176.471,15.531,152.022
C01454=1098.736,70.850,441.901,176.473,15.531,152.022
C01455=1098.742,71.100,441.884,176.476,15.532,152.022
C01456=1098.747,71.349,441.867,176.478,15.532,152.021
C01457=1098.753,71.598,441.850,176.481,15.533,152.021
C01458=1098.758,71.848,441.833,176.483,15.534,152.020
C01459=1098.764,72.097,441.817,176.486,15.533,152.020
C01460=1098.770,72.346,441.799,176.489,15.534,152.019
C01461=1098.776,72.597,441.782,176.491,15.535,152.019
C01462=1098.782,72.845,441.765,176.494,15.535,152.019
C01463=1098.787,73.095,441.748,176.496,15.536,152.018
C01464=1098.793,73.344,441.732,176.499,15.537,152.018
C01465=1098.799,73.593,441.714,176.501,15.537,152.017
C01466=1098.804,73.843,441.698,176.504,15.538,152.017
C01467=1098.810,74.092,441.681,176.506,15.538,152.017
C01468=1098.815,74.341,441.664,176.509,15.538,152.016
C01469=1098.821,74.590,441.646,176.511,15.539,152.016
C01470=1098.827,74.841,441.630,176.514,15.539,152.015
C01471=1098.833,75.090,441.612,176.517,15.540,152.015
C01472=1098.838,75.339,441.595,176.519,15.541,152.014
C01473=1098.844,75.588,441.578,176.522,15.542,152.014
C01474=1098.849,75.838,441.561,176.524,15.541,152.013
C01475=1098.855,76.087,441.544,176.526,15.542,152.013
C01476=1098.860,76.336,441.527,176.529,15.542,152.013
C01477=1098.867,76.586,441.510,176.532,15.543,152.012
C01478=1098.872,76.835,441.493,176.535,15.544,152.012
C01479=1098.878,77.084,441.475,176.537,15.544,152.011
C01480=1098.884,77.334,441.459,176.540,15.545,152.011
C01481=1098.889,77.583,441.441,176.542,15.545,152.010
C01482=1098.895,77.833,441.423,176.545,15.546,152.010
C01483=1098.901,78.082,441.406,176.547,15.546,152.009
C01484=1098.907,78.331,441.390,176.550,15.547,152.009
C01485=1098.912,78.581,441.373,176.553,15.547,152.009
C01486=1098.918,78.830,441.355,176.555,15.547,152.008
C01487=1098.923,79.079,441.338,176.558,15.548,152.008
C01488=1098.929,79.329,441.320,176.560,15.548,152.007
C01489=1098.935,79.602,441.301,176.563,15.549,152.007
C01490=1098.941,79.875,441.282,176.566,15.549,152.006
C01491=1098.948,80.149,441.263,176.569,15.550,152.006
C01492=1098.954,80.423,441.245,176.572,15.550,152.005
C01493=1098.959,80.672,441.227,176.575,15.551,152.005
C01494=1098.965,80.922,441.210,176.577,15.551,152.004
C01495=1098.971,81.171,441.192,176.579,15.551,152.004
C01496=1098.976,81.421,441.175,176.582,15.552,152.003
C01497=1098.981,81.670,441.158,176.584,15.553,152.003
C01498=1098.988,81.918,441.141,176.588,15.553,152.002
C01499=1098.993,82.169,441.123,176.590,15.553,152.002
C01500=1098.999,82.418,441.106,176.593,15.554,152.002
C01501=1099.005,82.667,441.088,176.595,15.554,152.001
C01502=1099.010,82.916,441.071,176.598,15.555,152.001
C01503=1099.016,83.166,441.053,176.600,15.555,152.000
C01504=1099.021,83.415,441.036,176.603,15.556,152.000
C01505=1099.027,83.664,441.018,176.606,15.556,151.999
C01506=1099.032,83.913,441.001,176.609,15.557,151.999
C01507=1099.039,84.163,440.983,176.611,15.557,151.998
C01508=1099.044,84.413,440.966,176.614,15.558,151.998
C01509=1099.049,84.662,440.948,176.617,15.558,151.997
C01510=1099.055,84.911,440.931,176.619,15.558,151.997
C01511=1099.061,85.160,440.913,176.622,15.559,151.997
C01512=1099.066,85.410,440.895,176.624,15.559,151.996
C01513=1099.072,85.659,440.878,176.627,15.560,151.996
C01514=1099.078,85.908,440.860,176.630,15.559,151.995
C01515=1099.084,86.158,440.844,176.633,15.560,151.995
C01516=1099.090,86.407,440.826,176.635,15.561,151.994
C01517=1099.096,86.656,440.808,176.638,15.561,151.994
C01518=1099.101,86.905,440.790,176.640,15.561,151.993
C01519=1099.107,87.155,440.773,176.643,15.562,151.993
C01520=1099.113,87.404,440.755,176.646,15.562,151.992
C01521=1099.118,87.653,440.737,176.649,15.563,151.992
C01522=1099.124,87.902,440.720,176.651,15.563,151.991
C01523=1099.130,88.152,440.702,176.654,15.564,151.991
C01524=1099.135,88.401,440.684,176.657,15.563,151.990
C01525=1099.141,88.650,440.667,176.660,15.564,151.990
C01526=1099.146,88.900,440.648,176.662,15.564,151.989
C01527=1099.152,89.149,440.631,176.664,15.564,151.989
C01528=1099.157,89.398,440.613,176.667,15.565,151.988
C01529=1099.164,89.648,440.595,176.670,15.565,151.988
C01530=1099.169,89.897,440.578,176.673,15.566,151.987
C01531=1099.175,90.147,440.560,176.675,15.566,151.987
C01532=1099.181,90.396,440.542,176.678,15.566,151.986
C01533=1099.186,90.645,440.525,176.681,15.567,151.986
C01534=1099.192,90.895,440.507,176.684,15.567,151.985
C01535=1099.198,91.144,440.489,176.686,15.567,151.985
C01536=1099.203,91.393,440.471,176.689,15.568,151.984
C01537=1099.210,91.642,440.454,176.691,15.568,151.984
C01538=1099.215,91.891,440.435,176.695,15.568,151.983
C01539=1099.221,92.141,440.417,176.697,15.569,151.983
C01540=1099.226,92.390,440.399,176.700,15.569,151.982
C01541=1099.232,92.639,440.382,176.702,15.569,151.982
C01542=1099.238,92.889,440.364,176.706,15.570,151.981
C01543=1099.243,93.138,440.346,176.708,15.570,151.981
C01544=1099.248,93.387,440.328,176.711,15.571,151.980
C01545=1099.254,93.637,440.310,176.713,15.571,151.980
C01546=1099.260,93.885,440.292,176.717,15.571,151.979
C01547=1099.265,94.135,440.273,176.719,15.572,151.979
C01548=1099.271,94.384,440.256,176.722,15.572,151.978
C01549=1099.277,94.633,440.238,176.724,15.572,151.978
C01550=1099.283,94.883,440.220,176.727,15.573,151.977
C01551=1099.288,95.132,440.201,176.730,15.573,151.977
C01552=1099.294,95.382,440.183,176.733,15.573,151.976
C01553=1099.300,95.656,440.163,176.735,15.573,151.976
C01554=1099.306,95.928,440.144,176.739,15.574,151.975
C01555=1099.312,96.203,440.124,176.742,15.574,151.974
C01556=1099.319,96.476,440.105,176.745,15.575,151.974
C01557=1099.324,96.725,440.086,176.747,15.575,151.973
C01558=1099.330,96.975,440.068,176.751,15.575,151.973
C01559=1099.336,97.224,440.050,176.753,15.575,151.972
C01560=1099.341,97.473,440.031,176.756,15.576,151.972
C01561=1099.347,97.722,440.013,176.759,15.576,151.971
C01562=1099.353,97.972,439.996,176.762,15.576,151.971
C01563=1099.358,98.221,439.977,176.764,15.577,151.970
C01564=1099.364,98.471,439.959,176.767,15.577,151.970
C01565=1099.370,98.720,439.941,176.770,15.577,151.969
C01566=1099.375,98.969,439.922,176.773,15.577,151.968
C01567=1099.381,99.218,439.904,176.775,15.578,151.968
C01568=1099.387,99.468,439.886,176.779,15.578,151.967
C01569=1099.392,99.717,439.868,176.781,15.578,151.967
C01570=1099.398,99.966,439.850,176.784,15.578,151.966
C01571=1099.404,100.215,439.831,176.787,15.579,151.966
C01572=1099.409,100.465,439.813,176.790,15.579,151.965
C01573=1099.415,100.713,439.795,176.792,15.579,151.965
C01574=1099.421,100.963,439.777,176.796,15.579,151.964
C01575=1099.427,101.213,439.758,176.798,15.580,151.964
C01576=1099.432,101.461,439.740,176.801,15.580,151.963
C01577=1099.438,101.712,439.721,176.804,15.580,151.963
C01578=1099.444,101.960,439.703,176.807,15.580,151.962
C01579=1099.449,102.210,439.684,176.809,15.581,151.962
C01580=1099.455,102.458,439.666,176.812,15.581,151.961
C01581=1099.460,102.708,439.648,176.815,15.581,151.960
C01582=1099.466,102.957,439.629,176.818,15.581,151.960
C01583=1099.471,103.207,439.611,176.820,15.581,151.959
C01584=1099.477,103.455,439.593,176.823,15.582,151.959
C01585=1099.483,103.705,439.574,176.826,15.582,151.958
C01586=1099.489,103.954,439.556,176.829,15.582,151.958
C01587=1099.494,104.203,439.537,176.832,15.582,151.957
C01588=1099.500,104.452,439.519,176.835,15.583,151.957
C01589=1099.505,104.702,439.500,176.837,15.583,151.956
C01590=1099.511,104.952,439.481,176.840,15.583,151.956
C01591=1099.517,105.200,439.463,176.843,15.583,151.955
C01592=1099.522,105.450,439.444,176.846,15.584,151.954
C01593=1099.528,105.699,439.426,176.849,15.583,151.954
C01594=1099.534,105.948,439.407,176.852,15.584,151.953
C01595=1099.540,106.198,439.389,176.854,15.584,151.953
C01596=1099.545,106.447,439.370,176.858,15.584,151.952
C01597=1099.550,106.696,439.351,176.861,15.585,151.951
C01598=1099.556,106.945,439.333,176.863,15.585,151.951
C01599=1099.562,107.194,439.314,176.866,15.585,151.950
C01600=1099.568,107.444,439.295,176.869,15.585,151.950
C01601=1099.573,107.693,439.277,176.872,15.586,151.949
C01602=1099.579,107.942,439.258,176.875,15.586,151.949
C01603=1099.585,108.191,439.239,176.878,15.586,151.948
C01604=1099.590,108.440,439.220,176.880,15.586,151.948
C01605=1099.596,108.690,439.202,176.884,15.586,151.947
C01606=1099.602,108.939,439.183,176.886,15.586,151.946
C01607=1099.607,109.188,439.164,176.889,15.587,151.946
C01608=1099.613,109.437,439.146,176.892,15.586,151.945
C01609=1099.619,109.687,439.127,176.895,15.587,151.945
C01610=1099.624,109.936,439.108,176.898,15.587,151.944
C01611=1099.630,110.185,439.090,176.901,15.587,151.944
C01612=1099.636,110.435,439.070,176.903,15.587,151.943
C01613=1099.641,110.683,439.052,176.907,15.587,151.942
C01614=1099.647,110.933,439.034,176.909,15.587,151.942
C01615=1099.653,111.183,439.014,176.913,15.587,151.941
C01616=1099.658,111.431,438.995,176.916,15.588,151.941
C01617=1099.665,111.705,438.974,176.919,15.588,151.940
C01618=1099.671,111.979,438.954,176.922,15.588,151.939
C01619=1099.677,112.253,438.933,176.925,15.588,151.939
C01620=1099.684,112.526,438.913,176.929,15.588,151.938
C01621=1099.689,112.776,438.893,176.931,15.588,151.937
C01622=1099.694,113.024,438.875,176.934,15.589,151.937
C01623=1099.700,113.274,438.855,176.937,15.589,151.936
C01624=1099.706,113.523,438.837,176.940,15.589,151.936
C01625=1099.712,113.772,438.817,176.943,15.588,151.935
C01626=1099.717,114.021,438.799,176.946,15.589,151.934
C01627=1099.723,114.270,438.779,176.949,15.589,151.934
C01628=1099.729,114.520,438.760,176.952,15.589,151.933
C01629=1099.734,114.768,438.742,176.954,15.589,151.933
C01630=1099.740,115.018,438.723,176.958,15.589,151.932
C01631=1099.745,115.268,438.704,176.961,15.590,151.932
C01632=1099.751,115.517,438.685,176.963,15.590,151.931
C01633=1099.756,115.766,438.666,176.967,15.590,151.930
C01634=1099.762,116.015,438.647,176.970,15.590,151.930
C01635=1099.768,116.264,438.627,176.973,15.590,151.929
C01636=1099.773,116.513,438.608,176.975,15.590,151.928
C01637=1099.779,116.762,438.589,176.979,15.590,151.928
C01638=1099.784,117.012,438.569,176.981,15.590,151.927
C01639=1099.790,117.261,438.550,176.984,15.591,151.927
C01640=1099.795,117.510,438.531,176.988,15.591,151.926
C01641=1099.801,117.759,438.512,176.990,15.590,151.925
C01642=1099.807,118.009,438.493,176.994,15.591,151.925
C01643=1099.812,118.258,438.474,176.996,15.591,151.924
C01644=1099.817,118.507,438.455,176.999,15.591,151.924
C01645=1099.823,118.756,438.435,177.002,15.591,151.923
C01646=1099.829,119.006,438.416,177.005,15.591,151.922
C01647=1099.835,119.255,438.396,177.008,15.591,151.922
C01648=1099.840,119.504,438.377,177.011,15.591,151.921
C01649=1099.845,119.753,438.358,177.014,15.592,151.921
C01650=1099.851,120.002,438.339,177.017,15.591,151.920
C01651=1099.857,120.252,438.320,177.021,15.592,151.919
C01652=1099.862,120.501,438.300,177.023,15.592,151.919
C01653=1099.868,120.750,438.280,177.027,15.592,151.918
C01654=1099.874,120.999,438.262,177.029,15.591,151.917
C01655=1099.879,121.248,438.242,177.032,15.592,151.917
C01656=1099.885,121.498,438.223,177.035,15.592,151.916
C01657=1099.891,121.746,438.203,177.038,15.592,151.916
C01658=1099.897,121.996,438.184,177.042,15.592,151.915
C01659=1099.902,122.245,438.165,177.044,15.592,151.914
C01660=1099.907,122.494,438.146,177.048,15.592,151.914
C01661=1099.913,122.743,438.126,177.050,15.592,151.913
C01662=1099.918,122.993,438.106,177.054,15.592,151.912
C01663=1099.924,123.242,438.087,177.056,15.592,151.912
C01664=1099.930,123.491,438.067,177.060,15.592,151.911
C01665=1099.936,123.740,438.047,177.062,15.592,151.911
C01666=1099.941,123.990,438.028,177.066,15.592,151.910
C01667=1099.947,124.238,438.008,177.069,15.592,151.909
C01668=1099.952,124.487,437.989,177.072,15.592,151.909
C01669=1099.958,124.737,437.970,177.075,15.592,151.908
C01670=1099.964,124.985,437.950,177.078,15.592,151.907
C01671=1099.970,125.235,437.931,177.081,15.592,151.907
C01672=1099.975,125.484,437.910,177.084,15.592,151.906
C01673=1099.981,125.733,437.891,177.087,15.592,151.905
C01674=1099.986,125.983,437.872,177.091,15.592,151.905
C01675=1099.992,126.232,437.852,177.093,15.592,151.904
C01676=1099.998,126.481,437.833,177.097,15.592,151.903
C01677=1100.004,126.730,437.813,177.099,15.592,151.903
C01678=1100.010,126.979,437.793,177.103,15.592,151.902
C01679=1100.015,127.228,437.773,177.105,15.592,151.901
C01680=1100.021,127.478,437.754,177.109,15.592,151.901
C01681=1100.027,127.751,437.732,177.112,15.592,151.900
C01682=1100.033,128.025,437.711,177.116,15.592,151.899
C01683=1100.039,128.299,437.689,177.119,15.591,151.899
C01684=1100.046,128.572,437.667,177.122,15.591,151.898
C01685=1100.052,128.822,437.648,177.126,15.592,151.897
C01686=1100.057,129.071,437.627,177.128,15.591,151.896
C01687=1100.063,129.320,437.608,177.132,15.592,151.896
C01688=1100.069,129.569,437.588,177.134,15.591,151.895
C01689=1100.075,129.818,437.568,177.138,15.591,151.894
C01690=1100.081,130.067,437.549,177.141,15.591,151.894
C01691=1100.086,130.316,437.529,177.144,15.591,151.893
C01692=1100.092,130.566,437.509,177.148,15.591,151.892
C01693=1100.098,130.815,437.489,177.150,15.591,151.892
C01694=1100.104,131.064,437.469,177.154,15.591,151.891
C01695=1100.109,131.313,437.450,177.156,15.590,151.890
C01696=1100.115,131.562,437.430,177.160,15.591,151.890
C01697=1100.121,131.811,437.410,177.163,15.591,151.889
C01698=1100.126,132.060,437.390,177.166,15.590,151.888
C01699=1100.132,132.309,437.370,177.169,15.591,151.888
C01700=1100.138,132.558,437.350,177.172,15.590,151.887
C01701=1100.143,132.808,437.331,177.176,15.590,151.886
C01702=1100.148,133.057,437.310,177.179,15.590,151.886
C01703=1100.154,133.306,437.290,177.182,15.590,151.885
C01704=1100.160,133.555,437.270,177.185,15.590,151.884
C01705=1100.165,133.804,437.250,177.188,15.590,151.884
C01706=1100.171,134.053,437.230,177.191,15.590,151.883
C01707=1100.177,134.302,437.210,177.194,15.589,151.882
C01708=1100.183,134.551,437.190,177.197,15.590,151.882
C01709=1100.188,134.801,437.170,177.201,15.590,151.881
C01710=1100.194,135.050,437.150,177.204,15.589,151.880
C01711=1100.199,135.299,437.129,177.207,15.589,151.879
C01712=1100.205,135.548,437.109,177.210,15.589,151.879
C01713=1100.211,135.797,437.089,177.213,15.589,151.878
C01714=1100.216,136.047,437.069,177.217,15.589,151.877
C01715=1100.222,136.296,437.049,177.220,15.588,151.877
C01716=1100.228,136.545,437.029,177.223,15.589,151.876
C01717=1100.234,136.793,437.009,177.226,15.588,151.875
C01718=1100.239,137.043,436.988,177.229,15.588,151.875
C01719=1100.245,137.291,436.968,177.233,15.588,151.874
C01720=1100.250,137.541,436.948,177.236,15.588,151.873
C01721=1100.256,137.791,436.928,177.239,15.588,151.873
C01722=1100.262,138.040,436.908,177.242,15.588,151.872
C01723=1100.268,138.289,436.888,177.245,15.588,151.871
C01724=1100.273,138.538,436.867,177.248,15.587,151.870
C01725=1100.279,138.787,436.847,177.252,15.587,151.870
C01726=1100.284,139.036,436.827,177.255,15.587,151.869
C01727=1100.289,139.285,436.806,177.258,15.587,151.868
C01728=1100.296,139.534,436.786,177.261,15.587,151.868
C01729=1100.301,139.783,436.765,177.264,15.587,151.867
C01730=1100.307,140.032,436.745,177.268,15.587,151.866
C01731=1100.313,140.281,436.725,177.271,15.587,151.865
C01732=1100.319,140.530,436.705,177.274,15.586,151.865
C01733=1100.324,140.779,436.684,177.278,15.586,151.864
C01734=1100.329,141.028,436.664,177.280,15.586,151.863
C01735=1100.336,141.278,436.643,177.284,15.586,151.862
C01736=1100.341,141.527,436.623,177.287,15.586,151.862
C01737=1100.346,141.776,436.602,177.290,15.585,151.861
C01738=1100.352,142.025,436.582,177.294,15.585,151.860
C01739=1100.357,142.274,436.562,177.296,15.585,151.860
C01740=1100.363,142.523,436.541,177.300,15.585,151.859
C01741=1100.370,142.772,436.520,177.304,15.585,151.858
C01742=1100.375,143.021,436.500,177.306,15.584,151.857
C01743=1100.380,143.270,436.479,177.310,15.584,151.857
C01744=1100.386,143.519,436.459,177.313,15.584,151.856
C01745=1100.392,143.793,436.436,177.316,15.584,151.855
C01746=1100.398,144.067,436.413,177.320,15.583,151.854
C01747=1100.404,144.340,436.391,177.324,15.584,151.854
C01748=1100.411,144.613,436.368,177.327,15.584,151.853
C01749=1100.416,144.863,436.348,177.331,15.584,151.852
C01750=1100.422,145.112,436.327,177.334,15.583,151.851
C01751=1100.427,145.361,436.306,177.338,15.583,151.850
C01752=1100.433,145.610,436.286,177.340,15.582,151.850
C01753=1100.439,145.859,436.265,177.344,15.582,151.849
C01754=1100.444,146.108,436.244,177.348,15.582,151.848
C01755=1100.450,146.358,436.224,177.350,15.582,151.848
C01756=1100.456,146.607,436.204,177.354,15.582,151.847
C01757=1100.462,146.855,436.182,177.357,15.581,151.846
C01758=1100.467,147.105,436.161,177.360,15.581,151.845
C01759=1100.473,147.354,436.141,177.364,15.581,151.845
C01760=1100.479,147.602,436.120,177.367,15.581,151.844
C01761=1100.484,147.851,436.100,177.370,15.581,151.843
C01762=1100.490,148.101,436.079,177.373,15.580,151.842
C01763=1100.496,148.350,436.057,177.377,15.580,151.842
C01764=1100.501,148.599,436.037,177.380,15.580,151.841
C01765=1100.507,148.849,436.016,177.383,15.579,151.840
C01766=1100.512,149.097,435.995,177.387,15.579,151.839
C01767=1100.518,149.346,435.975,177.390,15.579,151.839
C01768=1100.524,149.596,435.954,177.393,15.579,151.838
C01769=1100.530,149.844,435.933,177.397,15.578,151.837
C01770=1100.535,150.093,435.912,177.400,15.578,151.836
C01771=1100.541,150.342,435.891,177.403,15.578,151.836
C01772=1100.546,150.592,435.870,177.407,15.578,151.835
C01773=1100.552,150.840,435.849,177.410,15.577,151.834
C01774=1100.557,151.089,435.828,177.413,15.577,151.833
C01775=1100.563,151.339,435.807,177.417,15.577,151.832
C01776=1100.569,151.588,435.786,177.420,15.576,151.832
C01777=1100.574,151.837,435.765,177.424,15.576,151.831
C01778=1100.580,152.086,435.744,177.426,15.576,151.830
C01779=1100.585,152.335,435.723,177.430,15.576,151.830
C01780=1100.591,152.584,435.702,177.434,15.575,151.829
C01781=1100.597,152.833,435.681,177.437,15.575,151.828
C01782=1100.602,153.082,435.660,177.440,15.575,151.827
C01783=1100.609,153.331,435.638,177.444,15.575,151.826
C01784=1100.614,153.580,435.617,177.447,15.574,151.826
C01785=1100.619,153.829,435.596,177.450,15.574,151.825
C01786=1100.625,154.079,435.575,177.453,15.573,151.824
C01787=1100.631,154.327,435.554,177.457,15.573,151.823
C01788=1100.637,154.577,435.533,177.461,15.573,151.822
C01789=1100.642,154.825,435.512,177.463,15.573,151.822
C01790=1100.648,155.074,435.490,177.467,15.573,151.821
C01791=1100.654,155.324,435.470,177.471,15.572,151.820
C01792=1100.659,155.572,435.448,177.474,15.572,151.819
C01793=1100.665,155.821,435.427,177.477,15.572,151.819
C01794=1100.671,156.071,435.406,177.480,15.571,151.818
C01795=1100.676,156.319,435.385,177.484,15.571,151.817
C01796=1100.682,156.568,435.363,177.487,15.571,151.816
C01797=1100.688,156.817,435.343,177.490,15.570,151.815
C01798=1100.693,157.067,435.320,177.494,15.570,151.815
C01799=1100.699,157.315,435.299,177.498,15.570,151.814
C01800=1100.704,157.565,435.278,177.501,15.569,151.813
C01801=1100.710,157.814,435.257,177.504,15.569,151.812
C01802=1100.716,158.062,435.236,177.508,15.569,151.811
C01803=1100.722,158.311,435.214,177.511,15.568,151.811
C01804=1100.727,158.561,435.193,177.515,15.568,151.810
C01805=1100.732,158.810,435.171,177.518,15.567,151.809
C01806=1100.738,159.059,435.150,177.521,15.567,151.808
C01807=1100.744,159.308,435.128,177.525,15.567,151.807
C01808=1100.750,159.556,435.107,177.528,15.566,151.807
C01809=1100.756,159.830,435.084,177.532,15.566,151.806
C01810=1100.762,160.104,435.060,177.536,15.566,151.805
C01811=1100.768,160.377,435.037,177.539,15.565,151.804
C01812=1100.775,160.650,435.013,177.543,15.565,151.803
C01813=1100.780,160.898,434.991,177.547,15.565,151.802
C01814=1100.786,161.148,434.970,177.550,15.564,151.802
C01815=1100.791,161.397,434.949,177.554,15.564,151.801
C01816=1100.797,161.646,434.927,177.557,15.564,151.800
C01817=1100.803,161.895,434.906,177.560,15.563,151.799
C01818=1100.808,162.144,434.883,177.564,15.563,151.798
